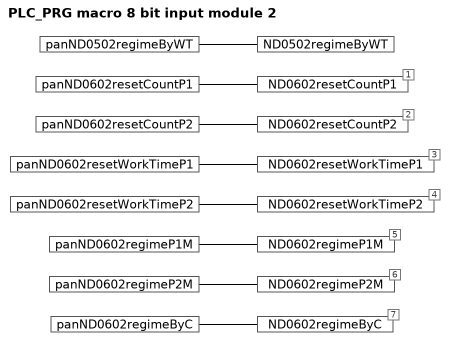
[picture p72: PLC_PRG macro 8 bit input module 2 (CFC)]
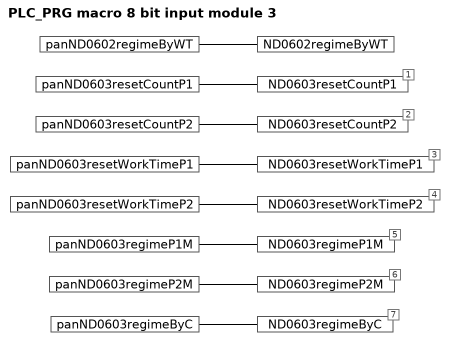
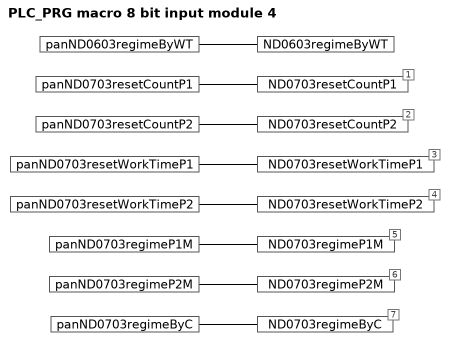
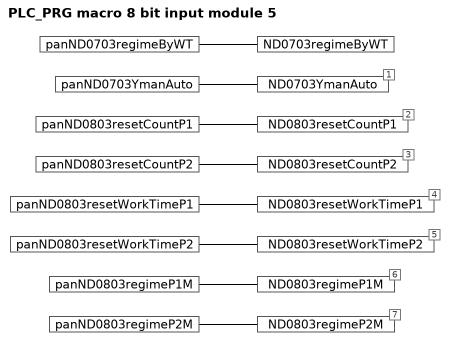
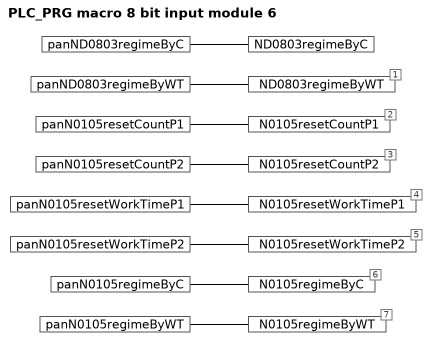
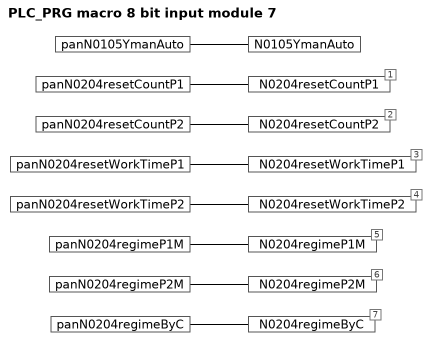
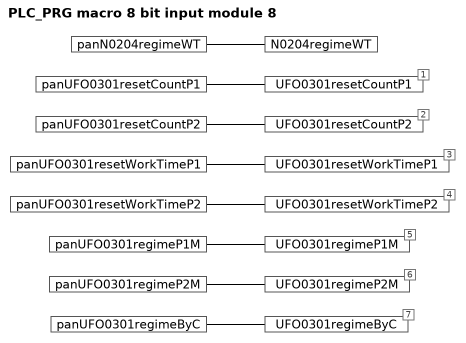
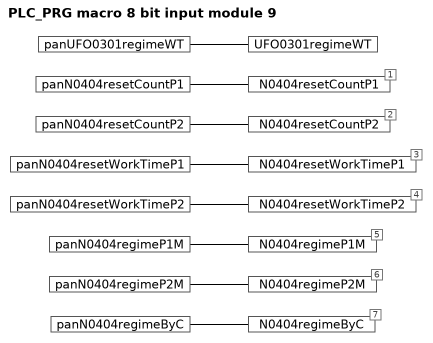
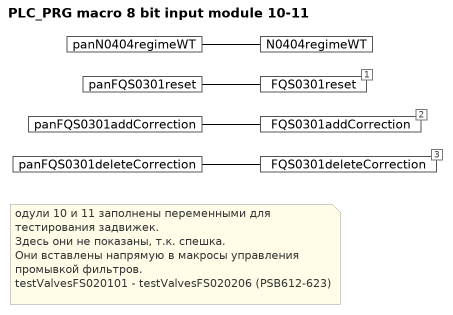
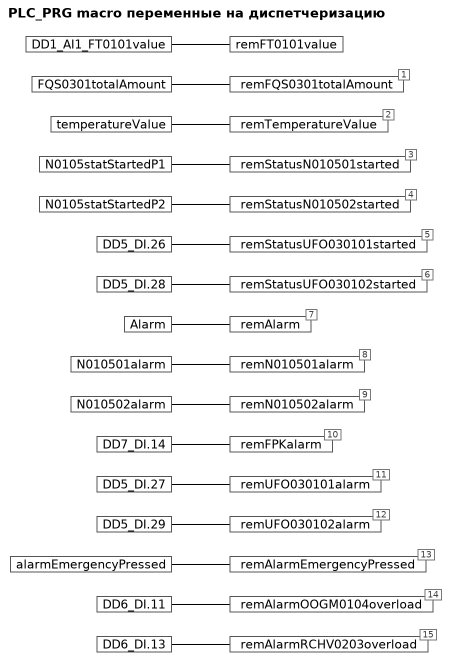
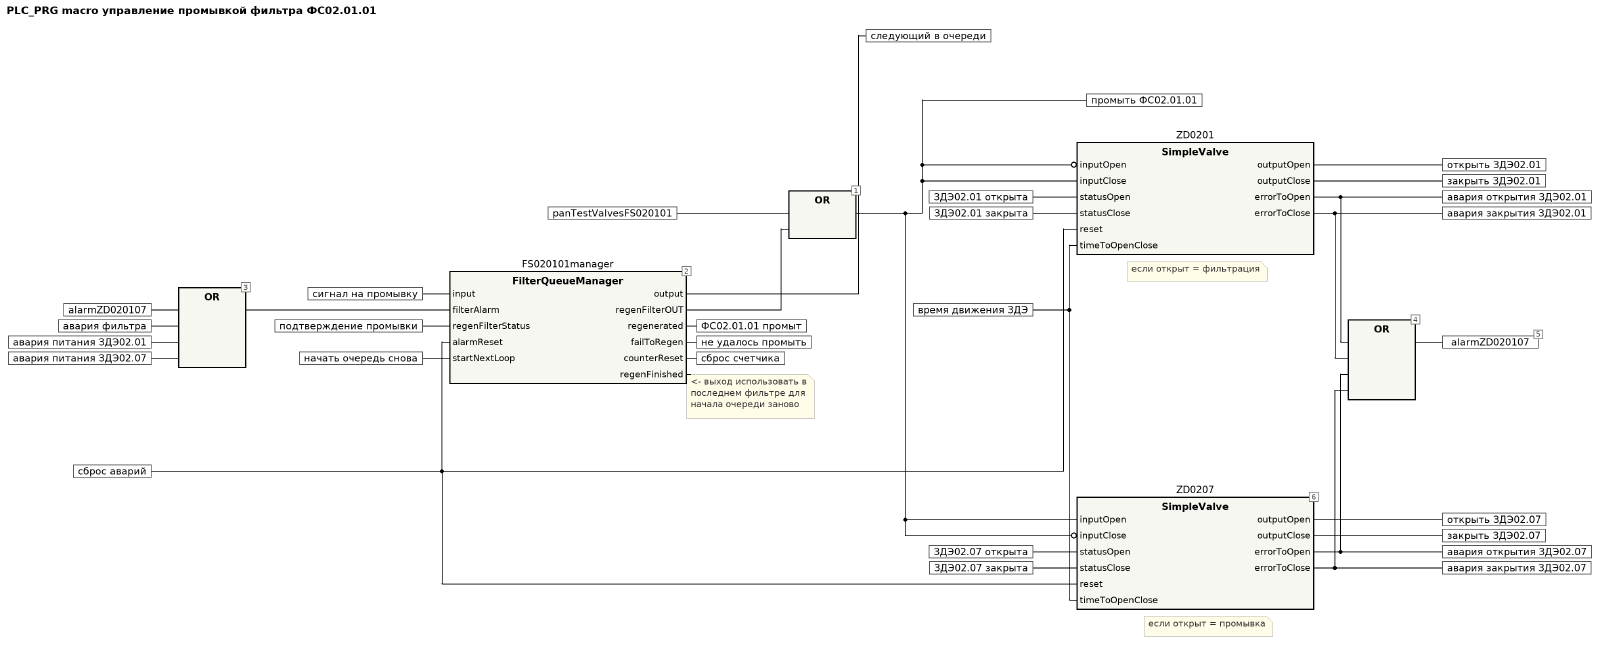
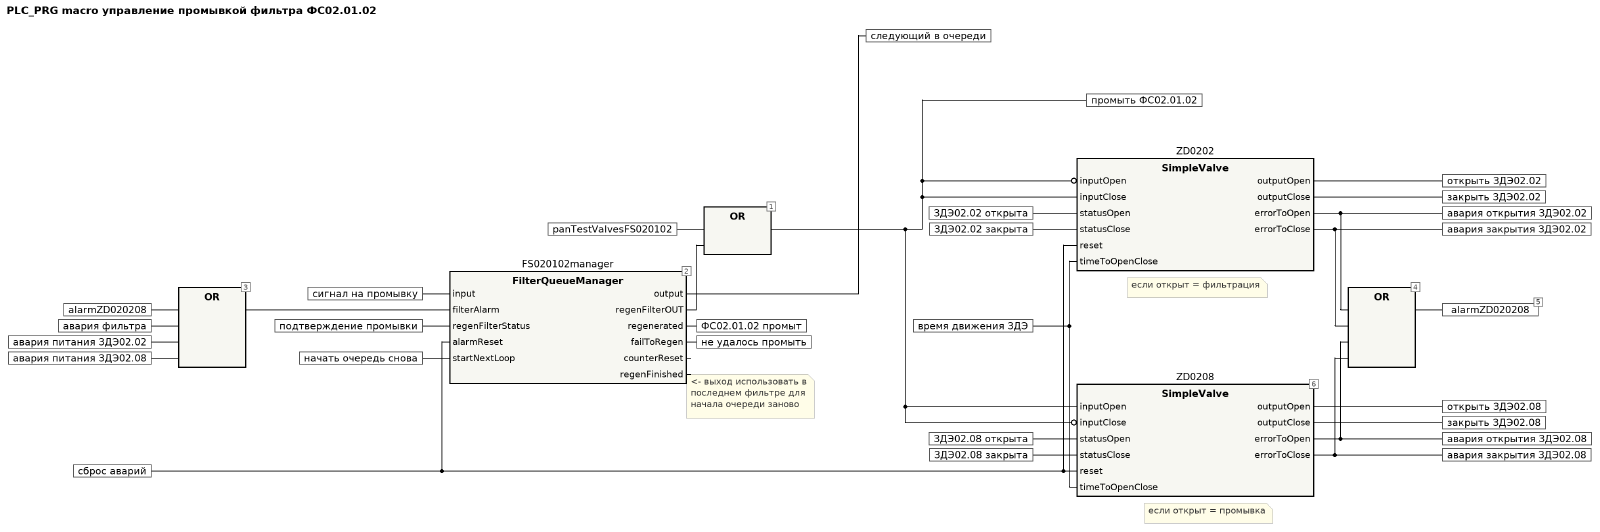
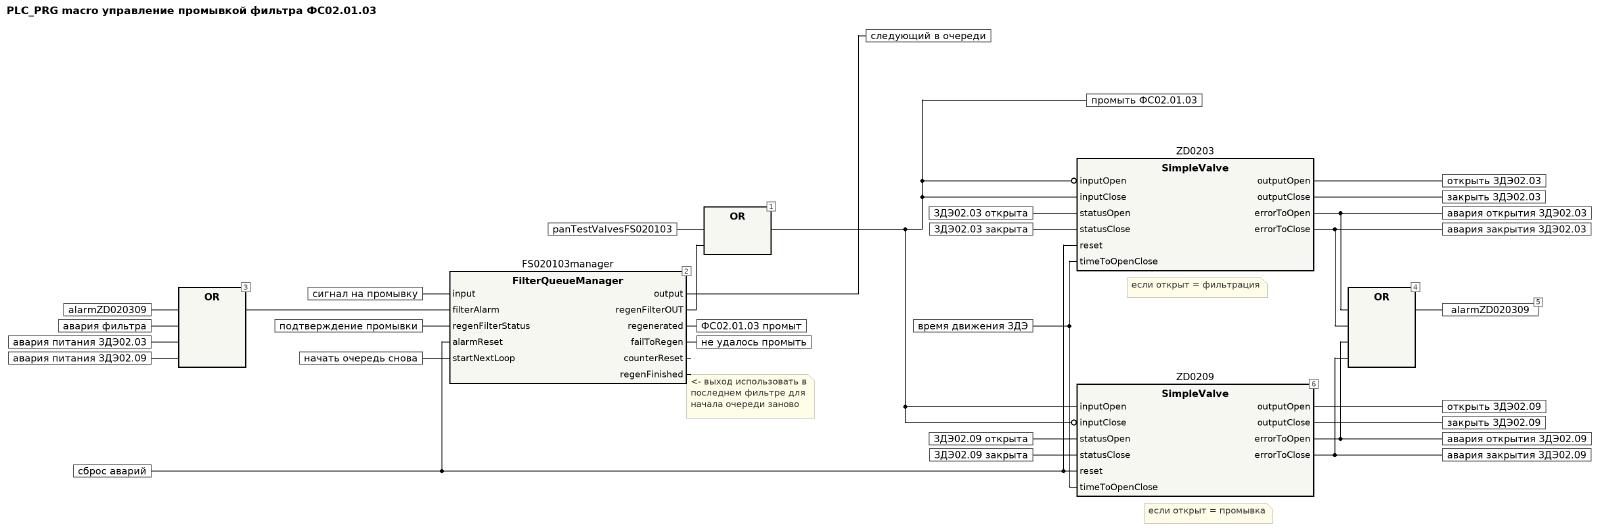
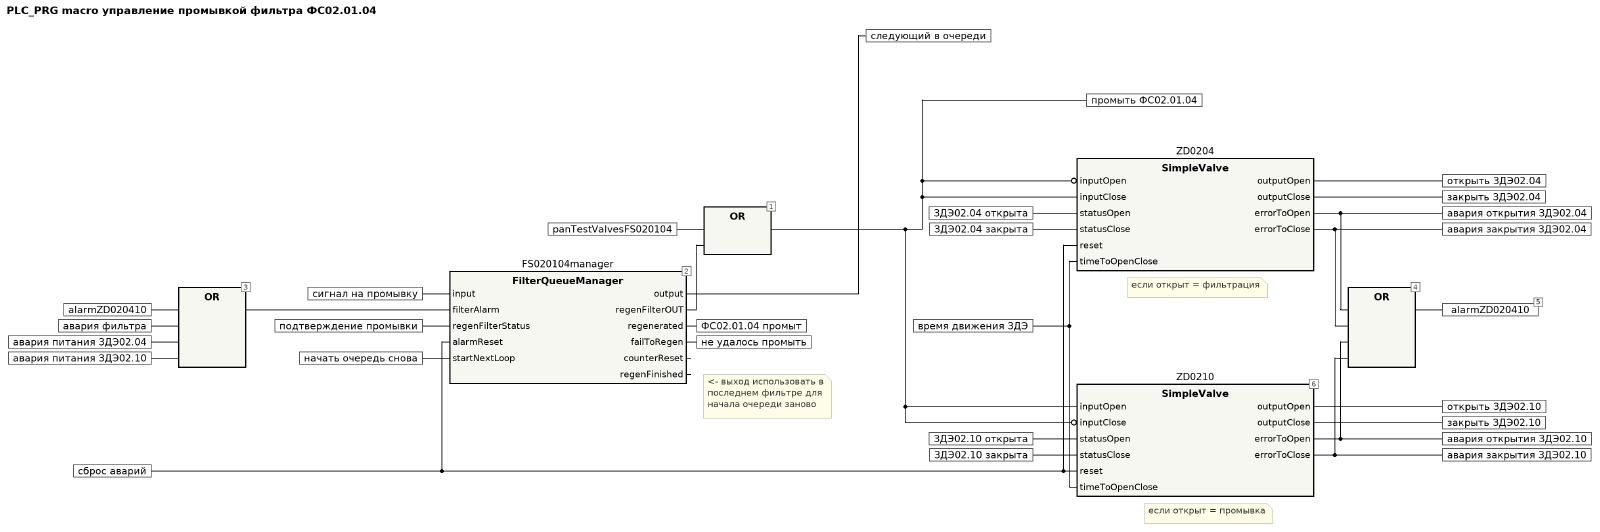
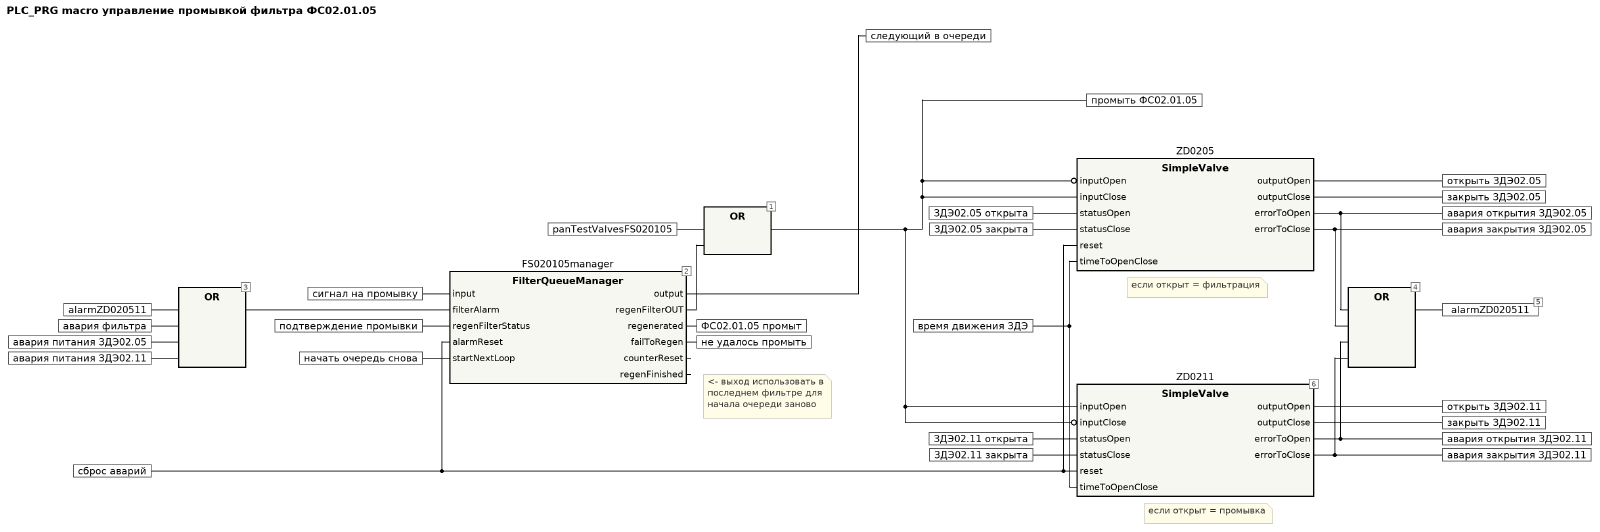
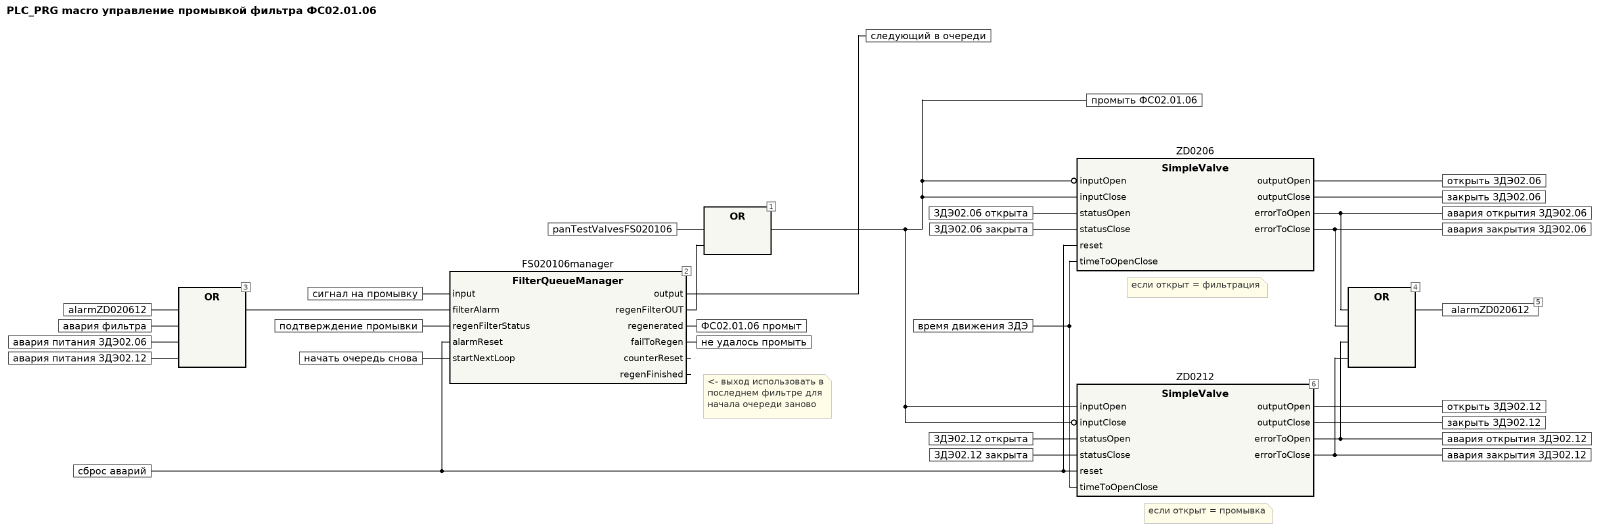
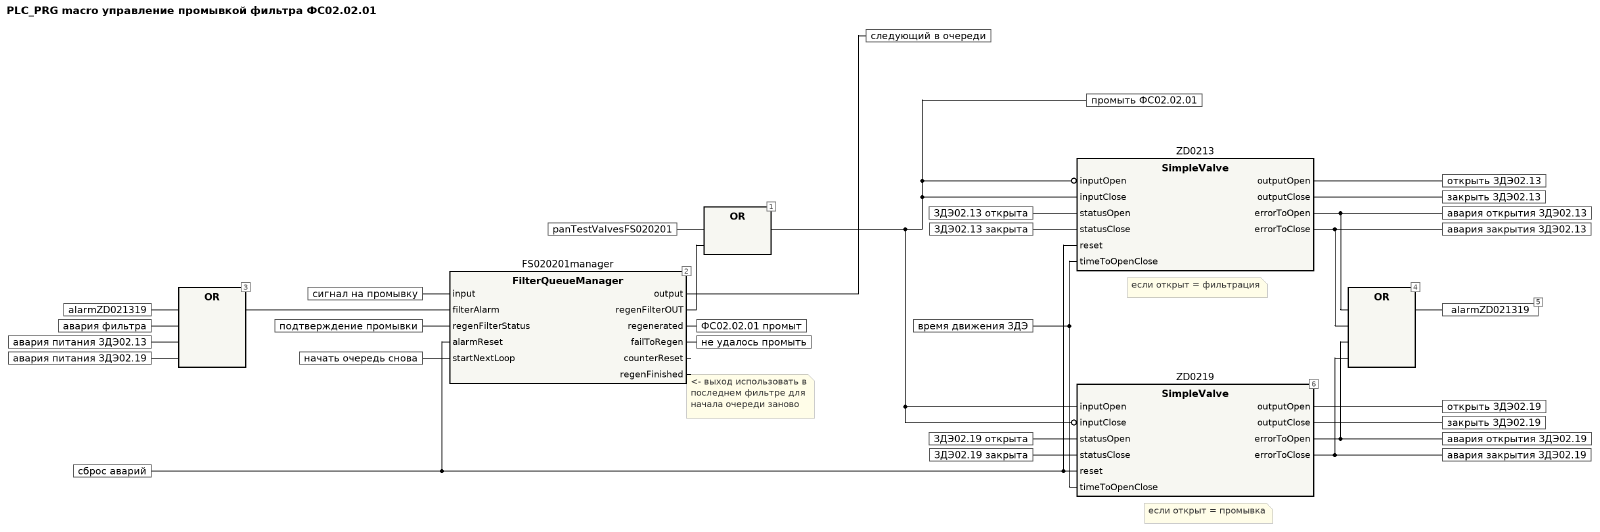
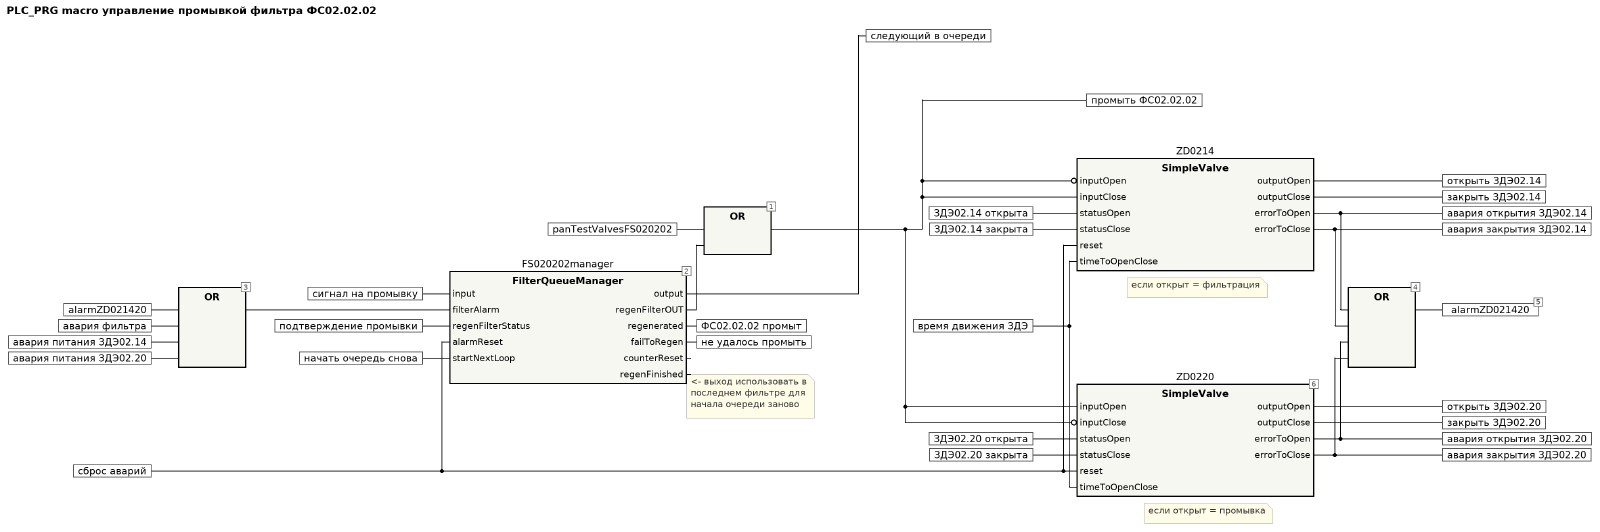
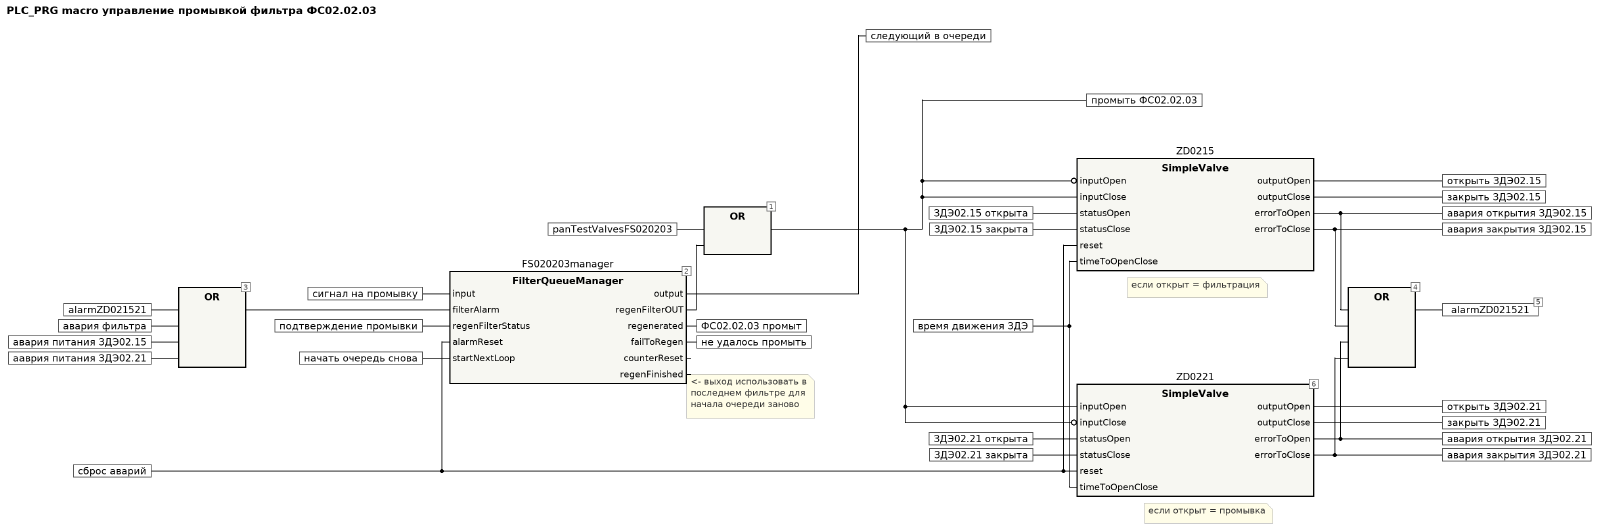
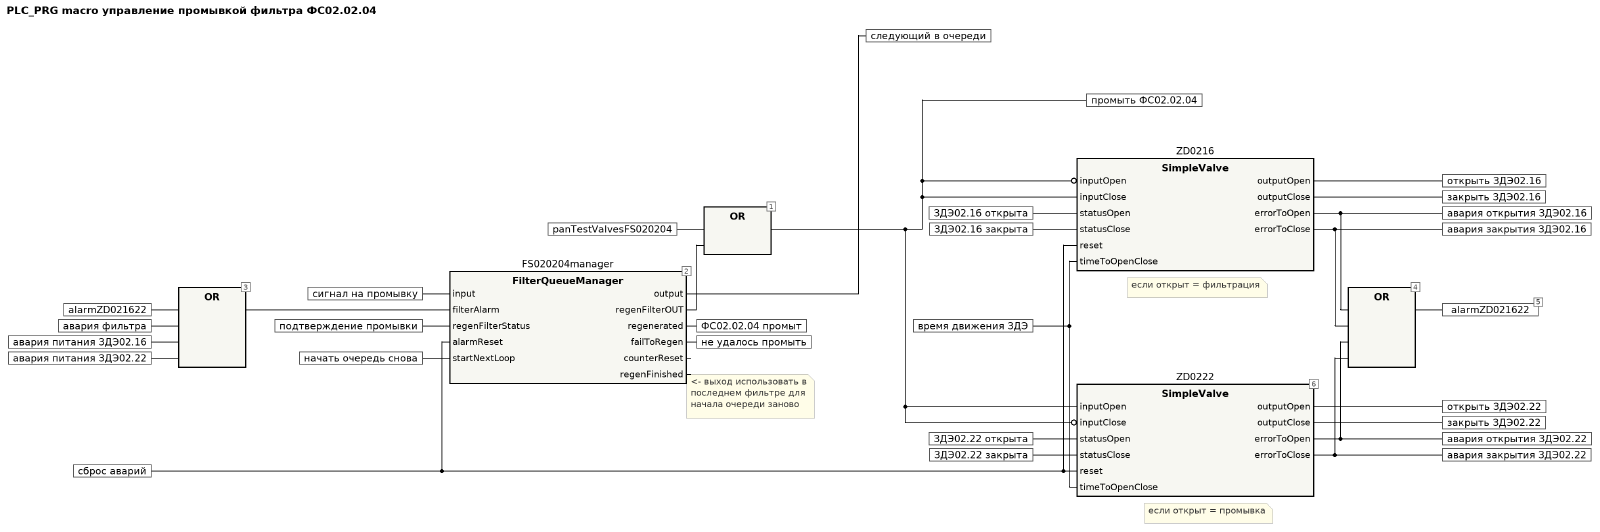
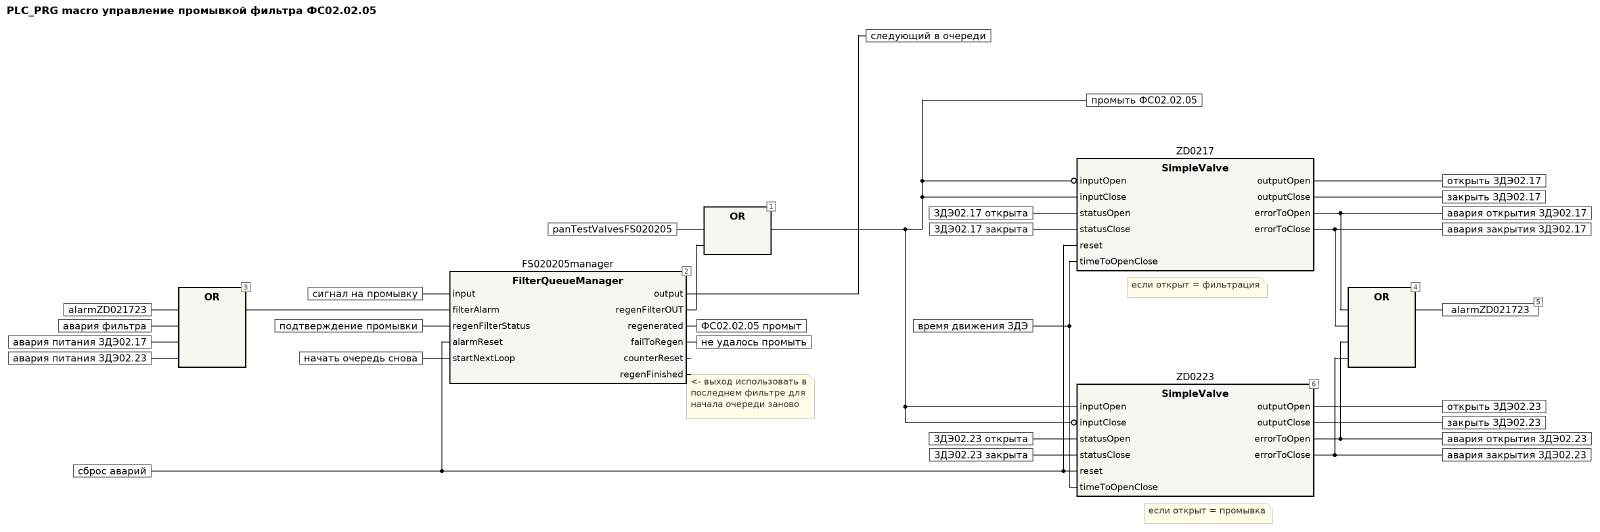
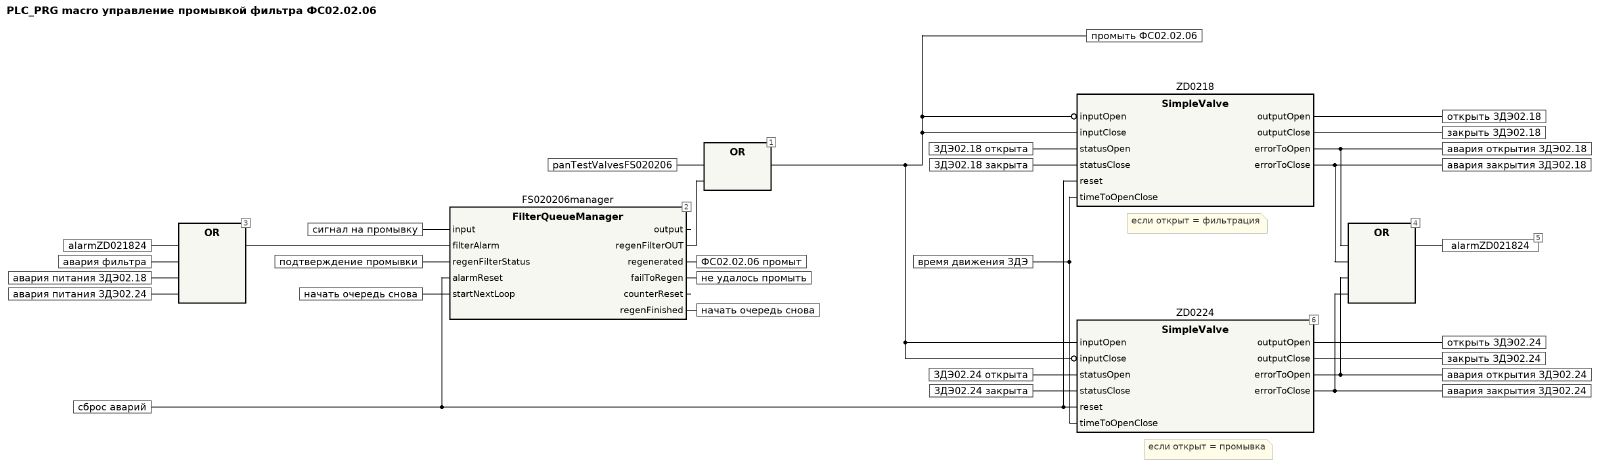
_CFC_ (* Continuous Function Chart, elements in execution order *)
(* в этом макросе лежит управление режимом тестирования задвижек ЗДЭ03 / Тестирование запрещает автоматический запуск УФО от ПЛК *)
(* 1=открыть; 0 = закрыть *)
(* авария питания КШЭ04.01 *)
(* авария НД05.02/02 *)
(* авария НД05.02/01 *)
(* инвертирование сигнала, чтобы все аварии / обозначались как 1 (TRUE) *)
(* авария питания ЗДЭ02.24 *)
(* авария питания ЗДЭ02.23 *)
(* авария питания ЗДЭ02.22 *)
(* авария питания ЗДЭ02.21 *)
(* авария питания ЗДЭ02.20 *)
(* авария питания ЗДЭ02.19 *)
(* авария питания ЗДЭ02.18 *)
(* авария питания ЗДЭ02.17 *)
(* авария питания ЗДЭ02.16 *)
(* авария питания ЗДЭ02.15 *)
(* авария питания ЗДЭ02.14 *)
(* авария питания ЗДЭ02.13 *)
(* авария питания ЗДЭ02.12 *)
(* авария питания ЗДЭ02.11 *)
(* авария питания ЗДЭ02.10 *)
(* авария питания ЗДЭ02.09 *)
(* авария питания ЗДЭ02.08 *)
(* авария питания ЗДЭ02.07 *)
(* авария питания ЗДЭ02.06 *)
(* авария питания ЗДЭ02.05 *)
(* авария питания ЗДЭ02.04 *)
(* авария питания ЗДЭ02.03 *)
(* авария питания ЗДЭ02.02 *)
(* авария питания ЗДЭ02.01 *)
(* очередь передается на 2 ступень *)
(* подсчет общего объема стоков, прошедшего через расходомер FT01.02 *)
(* сброс счетчика стоков до следующей промывки *)
(* авария (при 0) ФС02.02/01 *)
(* авария (при 0) ФС02.02/02 *)
(* авария (при 0) ФС02.02/03 *)
(* авария (при 0) ФС02.02/04 *)
(* авария (при 0) ФС02.02/05 *)
(* авария (при 0) ФС02.02/06 *)
(* авария (при 0) ФС02.01/01 *)
(* авария (при 0) ФС02.01/02 *)
(* авария (при 0) ФС02.01/03 *)
(* авария (при 0) ФС02.01/04 *)
(* авария (при 0) ФС02.01/05 *)
(* авария (при 0) ФС02.01/06 *)
(* 0=авария *)
(* заданный до промывки объем *)
(* текущий объем *)
(* Пуск Н02.04/02 *)
(* Пуск Н02.04/01 *)
(* Стоп Н02.04 *)
(* Сухой ход Н02.04 (LS02.03) 0=сух.ход *)
(* Клапан КЭМ08.01 открыт. *)
(* Клапан КЭМ07.01 открыт. *)
(* Клапан КЭМ06.01 открыт. *)
(* Клапан КЭМ05.01 открыт. *)
(* промывка ФС02.02/01 *)
(* промывка ФС02.02/02 *)
(* промывка ФС02.02/03 *)
(* промывка ФС02.02/04 *)
(* промывка ФС02.02/05 *)
(* промывка ФС02.02/06 *)
(* Авария Н02.04/02 (0=авария) *)
(* Авария Н02.04/01 (0=авария) *)
(* импульсный расходомер *)
(* авария Н04.04/02, 0=авария *)
(* авария Н04.04/01, 0=авария *)
(* сухой ход Н04.04, 0=защита *)
(* авт.пуск Н04.04 *)
(* пуск Н04.04/01 *)
(* пуск Н04.04/02 *)
(* стоп Н04.04 *)
(* подающий насос ФПК работает *)
(* статус КШЭ04.01 закрыт *)
(* Закрыть КШЭ04.01 *)
(* статус КШЭ04.01 открыт *)
(* Открыть КШЭ04.01 *)
(* авария ФПК *)
(* Авария входа AI6 ПЛК, давл.ФПК *)
(* Давление на входе ФПК / 0...16 бар (мах допуст.10) *)
(* LSА02.01 Перелив РЧВ02.03 *)
(* авария питания ЗДЭ02.25 *)
(* термоконтакт Н01.05/02 *)
(* термоконтакт Н01.05/01 *)
(* Авария ЧРП Н01.05 *)
(* КМ3 питание насоса 2 *)
(* КМ2 питание насоса 1 *)
(* КМ1 питание ЧРП *)
(* Пуск  Н01.05 *)
(* время на создание потока *)
(* Стоп  Н01.05 (сброс самоподхвата реле) *)
(* SA1 Ручной выбор Н01.05/02 = главный *)
(* SA1 Ручной выбор Н01.05/01 = главный *)
(* LS01.04 - нижний уровень ОГМ01.04, сухой ход Н01.05 *)
(* LS01.03 - рабочий верхний уровень ОГМ01.04 автоматический пуск 01.05 *)
(* Статус ПУСК ЧРП Н01.05 *)
(* Инициализирует требуемые булевые переменные / в момент старта выполнения программы. *)
(* LSA01.02 перелив ОГМ01.04 *)
(* сухой ход НД08.03/02 *)
(* сухой ход НД08.03/01 *)
(* сухой ход НД08.03/02 *)
(* сухой ход НД08.03/01 *)
(* авария входа рН-метра QE01.02 *)
(* рН-метр QE01.01 на входе, / диапазон 0...14 *)
(* расходомер FT01.02 на входе, / диапазон 0...600куб/час *)
(* авария входа расходомера FT01.01 *)
(* управление 4...20мА НД08.04 *)
(* пуск/стоп НД08.04 *)
(* насос Н04.01 работает *)
(* авария НД08.04 *)
(* авария привода НД08.03/02 *)
(* авария привода НД08.03/01 *)
(* АВАРИИ *)
(* управление 4...20мА НД05.02/02 *)
(* пуск/стоп НД05.02/02 *)
(* авария НД05.02/02 *)
(* авария НД05.02/01 *)
(* пуск/стоп НД05.02/01 *)
(* управление 4...20мА НД05.02/01 *)
(* датчик температуры в помещении / (метран) диапазон: 0...+100С *)
(* лампа АВАРИЯ *)
(* авария входа датчика температуры *)
(* ошибка блока дозирования НД05.02 *)
(* авария НД06.02/02 *)
(* авария НД06.02/01 *)
(* управление 4...20мА НД06.02/02 *)
(* пуск/стоп НД06.02/02 *)
(* пуск/стоп НД06.02/01 *)
(* управление 4...20мА НД06.02/01 *)
(* авария НД06.03/02 *)
(* авария НД06.03/01 *)
(* управление 4...20мА НД06.03/02 *)
(* пуск/стоп НД06.03/02 *)
(* пуск/стоп НД06.03/01 *)
(* управление 4...20мА НД06.03/01 *)
(* авария НД06.02/02 *)
(* авария НД06.02/01 *)
(* авария НД06.03/02 *)
(* авария НД06.03/01 *)
(* авария НД07.03/02 *)
(* авария НД07.03/01 *)
(* пуск/стоп НД07.03/02 *)
(* пуск/стоп НД07.03/01 *)
(* управление 4...20мА НД07.03/02 *)
(* управление 4...20мА НД07.03/01 *)
(* авария НД07.03/02 *)
(* авария НД07.03/01 *)
(* авария привода НД08.03/02 *)
(* авария привода НД08.03/01 *)
(* управление 4...20мА НД08.03/02 *)
(* пуск/стоп НД08.03/02 *)
(* пуск/стоп НД08.03/01 *)
(* управление 4...20мА НД08.03/01 *)
(* авария НД08.04 *)
(* расходомер FT01.01 на входе, / диапазон 0...600куб/час *)
(* авария входа расходомера FT01.02 *)
(* авария входа рН-метра QE01.01 *)
(* рН-метр QE01.02 на входе, / диапазон 0...14 *)
(* ФПК не запустился *)
(* ФПК готов к приему *)
(* подающий насос ФПК работает *)
(* авария ФПК *)
(* Давление на входе ФПК (0...16 бар) *)
(* датчик уровня осадка *)
(* Защита от сухого хода насоса ФПК *)
(* запуск фильтрации *)
(* время работы ФПК после спада сигнала датч.осадка *)
(* время контроля старта ФПК (по умолч.=3мин) *)
(* авария Н04.04/02 *)
(* авария Н04.04/01 *)
(* авария УФО03.01/01 *)
(* авария УФО03.01/02 *)
(* работа УФО03.01/01 *)
(* Для подачи предостережения на пульте / оператора (при необходимости), а также / сигнализации лампой АВАРИЯ. *)
(* авария УФО03.01/01 *)
(* работа УФО03.01/02 *)
(* авария УФО03.01/02 *)
(* Контроль, если УФО включили вручную, / а потока при этом нет. *)
(* работа М06.04 (УПК) *)
(* работа М07.02 (УПЩ) *)
(* работа М08.02 (УПФ) *)
(* авария М06.04 (УПК) *)
(* авария М07.02 (УПЩ) *)
(* авария М08.02 (УПФ) *)
(* пуск/стоп НД07.03/02 *)
(* пуск/стоп НД07.03/01 *)
(* пуск/стоп НД08.04 *)
(* пуск/стоп НД06.02/02 *)
(* пуск/стоп НД06.02/01 *)
(* пуск/стоп НД06.03/02 *)
(* пуск/стоп НД06.03/01 *)
(* пуск/стоп НД08.03/02 *)
(* пуск/стоп НД08.03/01 *)
(* промывка ФС02.01/01 *)
(* промывка ФС02.01/02 *)
(* промывка ФС02.01/03 *)
(* промывка ФС02.01/04 *)
(* промывка ФС02.01/05 *)
(* промывка ФС02.01/06 *)
(* Авария Н02.04/02 (0=авария) *)
(* Авария Н02.04/01 (0=авария) *)
(* здесь мгновенный расход / в кубометрах в час (FT01.02) *)
(* выдает импульс / каждую секунду *)
(* если есть расход / (больше нуля) *)
(* преобразуем расход из / кубометров в час в / кубометры в секунду *)
(* суммируем каждую секунду значение / мгновенного расхода в кубометрах в секунду *)
(* блок подачи сигнала на промывку *)
(* авария КНС *)
(* Авария питания розеток / управл.клапанов фильтров. *)
(* Авария питания клапанов КЭМ. *)
(* авария сети (РКФ) *)
(* Блок управления разрешением работы КНС *)
(* Нажат аварийный стоп. *)
(* разрешение работы КНС / 1 = разрешено *)
(* авария сети (РКФ) *)
(* Нажат аварийный стоп. *)
(* LSA01.02 перелив ОГМ01.04 *)
(* контроль обрыва или ошибок модулей в сети ПЛК *)
(* вкл КМ2 *)
(* статус-пуск Н01.05/01 *)
(* Статус ПУСК / ЧРП Н01.05 *)
(* вкл КМ3 *)
(* статус-пуск Н01.05/02 *)
(* авария питания ЗДЭ03.01 *)
(* авария питания ЗДЭ03.02 *)
(* авария обоих УФО, если проблемы / открытия/закрытия на одной из задвижек *)
(* 0 = перелив *)
#0 rTrigStartInitializer:R_TRIG(CLK: TRUE)
#1 startInitializer <= #0.Q
#2 MACRO контроль температуры в помещении(pin 1 "вход датчика температуры": DD1_AI0, pin 2 "минимально допустимая температура в помещении": maxTemperature, pin 3 "максимально допустимая температура в помещении": minTemperature)
	(* не смотрим конкретный тип ошибки / (работает не точно, обрыв определяет как слишком маленькое значение) / если не равно 0 - значит на входе ошибка *)
	(* задаем границы допустимой температуры в помещении / проверяем что измеренное значение в заданном диапазоне *)
	#3 DD1_AI0_temperature:DECODE_FLOAT(VALUE: pin 1, DEF_VALUE: -)
	#4 NE(#3._ERR, 0)
	out 2 "авария датчика температуры" <= #4
	out 1 "температура в помещении" <= #3.OUT_VALUE
	#5 REAL_TO_INT(#3.OUT_VALUE)
	#6 temperatureLimits:LIMITALARM(IN: #5, HIGH: pin 3, LOW: pin 2)
	out 3 "температура выше заданного диапазона" <= #6.O
	out 4 "температура ниже заданного диапазона" <= #6.U
	#7 temperatureLimits:LIMITALARM(IN: -, HIGH: -, LOW: -)
END_MACRO
#8 temperatureValue <= #2.out 1
#9 DD1_AI0_error <= #2.out 2
#10 alarmHighTemperature <= #2.out 3
#11 alarmLowTemperature <= #2.out 4
#12 OR(testKSHE0401, DD7_DI.13)
#13 MACRO клапан шаровый перед ФПК (КШЭ04.01)(pin 1 "сигнал "подающий насос ФПК" работает": #12, pin 2 "статус КШЭ04.01 открыт": DD9_DI.2, pin 3 "статус КШЭ04.01 закрыт": DD9_DI.3, pin 4 "сброс аварий": alarmReset, pin 5 "время на открытие/закрытие": timeToOpenCloseValve)
	#14 FPKkshe0401DelayToOpen:TON(IN: #16.outputOpen, PT: T#1s)
	out 1 "выход на открытие КШЭ04.01" <= #14.Q
	#15 FPKkshe0401DelayToClose:TON(IN: #16.outputClose, PT: T#1s)
	out 2 "выход на закрытие КШЭ04.01" <= #15.Q
	#16 FPKkshe0401:SimpleValve(inputOpen: pin 1, inputClose: #17, statusOpen: pin 2, statusClose: pin 3, reset: pin 4, timeToOpenClose: pin 5)
	#17 NOT(pin 1)
	out 3 "авария на открытие КШЭ04.01" <= #16.errorToOpen
	out 4 "авария на закрытие КШЭ04.01" <= #16.errorToClose
END_MACRO
#18 DD4_DO.2 <= #13.out 1
#19 DD4_DO.3 <= #13.out 2
#20 FPKkshe0401errorToOpen <= #13.out 3
#21 FPKkshe0401errorToClose <= #13.out 4
#22 OR(DD1_AI0_error, DD1_AI1_error, DD1_AI2_error, DD1_AI3_error, DD1_AI4_error, alarmHighTemperature, alarmLowTemperature, ND0502dosingError, ND0602dosingError, ND0603dosingError, ND0803dosingError, ND0804dosingError, DD1_DI6, DD1_DI7, N010501alarm, N010502alarm, ZDE0225errorToOpen, ZDE0225errorToClose, DD7_DI.14, FPKnotStarted, DD1_AI5_error, FPKkshe0401errorToOpen, FPKkshe0401errorToClose, DD5_DI.27, DD5_DI.29, filterFailToRegen020101, errorToOpenZD0201, errorToCloseZD0201, errorToOpenZD0207, errorToCloseZD0207, filterFailToRegen020102, errorToOpenZD0202, errorToCloseZD0202, errorToOpenZD0208, errorToCloseZD0208, filterFailToRegen020103, errorToOpenZD0203, errorToCloseZD0203, errorToOpenZD0209, errorToCloseZD0209, filterFailToRegen020104, errorToOpenZD0204, errorToCloseZD0204, errorToOpenZD0210, errorToCloseZD0210, filterFailToRegen020105, errorToOpenZD0205, errorToCloseZD0205, errorToOpenZD0211, errorToCloseZD0211, filterFailToRegen020106, errorToOpenZD0206, errorToCloseZD0206, errorToOpenZD0212, errorToCloseZD0212, filterFailToRegen020201, errorToOpenZD0213, errorToCloseZD0213, errorToOpenZD0219, errorToCloseZD0219, filterFailToRegen020202, errorToOpenZD0214, errorToCloseZD0214, errorToOpenZD0220, errorToCloseZD0220, filterFailToRegen020203, errorToOpenZD0215, errorToCloseZD0215, errorToOpenZD0221, errorToCloseZD0221, filterFailToRegen020204, errorToOpenZD0216, errorToCloseZD0216, errorToOpenZD0222, errorToCloseZD0222, filterFailToRegen020205, errorToOpenZD0217, errorToCloseZD0217, errorToOpenZD0223, errorToCloseZD0223, filterFailToRegen020206, errorToOpenZD0218, errorToCloseZD0218, errorToOpenZD0224, errorToCloseZD0224, alarmPLKnetwork, alarmND050201, alarmND050202, alarmND060201, alarmND060202, alarmND060301, alarmND060302, alarmND070301, alarmND070302, alarmND080301, alarmND080302, alarmND0804, alarmOGM0104overload, alarmRCHV0203overload, alarmN040402, alarmN040401, alarmM0604, alarmM0702, alarmM0802, alarmN020401, alarmN020402, alarmFS020101, alarmFS020102, alarmFS020103, alarmFS020104, alarmFS020105, alarmFS020106, alarmFS020201, alarmFS020202, alarmFS020203, alarmFS020204, alarmFS020205, alarmFS020206, alarmZDE0201power, alarmZDE0202power, alarmZDE0203power, alarmZDE0204power, alarmZDE0205power, alarmZDE0206power, alarmZDE0207power, alarmZDE0208power, alarmZDE0209power, alarmZDE0210power, alarmZDE0211power, alarmZDE0212power, alarmZDE0213power, alarmZDE0214power, alarmZDE0215power, alarmZDE0216power, alarmZDE0217power, alarmZDE0218power, alarmZDE0219power, alarmZDE0220power, alarmZDE0221power, alarmZDE0222power, alarmZDE0223power, alarmZDE0224power, alarmZDE0225power, alarmKSHE0401power, alarmKNS, alarmPowerSocketFS, alarmKEMvalvesPower, alarmEmergencyPressed, alarmRKF, errorToOpenZDE0301, errorToCloseZDE0301, errorToOpenZDE0302, errorToCloseZDE0302, alarmZDE0301power, alarmZDE0302power)
#23 DD1_DO11 <= #22
#24 alarm <= #22
#25 MACRO контроль аналогового входа DD1_AI1(pin 1 "вход": DD1_AI1)
	(* Не смотрим конкретную ошибку, / определяем,что вход неисправен без расшифровки. *)
	#26 DD1_AI1_FT0101:DECODE_FLOAT(VALUE: pin 1, DEF_VALUE: -)
	#27 NE(#26._ERR, 0)
	out 2 "авария" <= #27
	out 1 "выход" <= #26.OUT_VALUE
END_MACRO
#28 DD1_AI1_FT0101value <= #25.out 1
#29 DD1_AI1_error <= #25.out 2
#30 MACRO контроль аналогового входа DD1_AI2(pin 1 "вход": DD1_AI2)
	(* Не смотрим конкретную ошибку, / определяем,что вход неисправен без расшифровки. *)
	#31 DD1_AI2_FT0102:DECODE_FLOAT(VALUE: pin 1, DEF_VALUE: -)
	#32 NE(#31._ERR, 0)
	out 2 "авария" <= #32
	out 1 "выход" <= #31.OUT_VALUE
END_MACRO
#33 DD1_AI2_FT0102value <= #30.out 1
#34 DD1_AI2_error <= #30.out 2
#35 MACRO управление Н01.05 (поддержание заданного расхода по FT01.02)(pin 1 "статус ПУСК ЧРП (реле)": DD5_DI.4, pin 2 "LS01.03 раб.уров.": DD6_DI.12, pin 3 "LS01.04 ниж.уров.(сух.ход)": DD5_DI.0, pin 4 "SA1ручной выб.Н01.05/01-главный": DD5_DI.5, pin 5 "SA1ручной выб.Н01.05/02-главный": DD5_DI.6, pin 6 "включить режим "по кол.вкл."": N0105regimeByC, pin 7 "включить режим "по наработке"": N0105regimeByWT, pin 8 "значение расхода от FT01.02": DD1_AI2_FT0102value, pin 9 "уставка расхода": N0105flowSetValue, pin 10 "время на создание потока": N0105minFlowTime, pin 11 "Р-коэфф.": N0105koeffP, pin 12 "I-коэфф": N0105koeffI, pin 13 "Д-коэфф": N0105koeffD, pin 14 "управление ЧРП в ручн.реж.(4...20мА)": N0105YoutManual, pin 15 "переключатель управление ЧРП РУЧН/АВТ": N0105YmanAuto, pin 16 "мин.допустимый расход": N0105minFlow, pin 17 "термоконтакт Н01.05/01": DD5_DI.2, pin 18 "термоконтакт Н01.05/02": DD5_DI.3, pin 19 "авария ЧРП Н01.05": DD5_DI.1, pin 20 "сброс аварии": alarmReset, pin 21 "сброс кол-ва вкл.Н01.05/01": N0105resetCountP1, pin 22 "сброс кол-ва вкл.Н01.05/02": N0105resetCountP2, pin 23 "сброс наработки Н01.05/01": N0105resetWorkTimeP1, pin 24 "сброс наработки Н01.05/02": N0105resetWorkTimeP2)
	(* Если насос создает давление меньше / указанного, то авария. *)
	(* если на входе true / то нижнее значение, / иначе то, что посередине *)
	(* по умолчанию при старте программы *)
	(* управление Н01.05 - поддержание / заданного расхода по FT01.02 *)
	(* режимы по количеству включений,  или по наработке / активны если оба входа SA1 не активны *)
	(* Пуск  Н01.05 *)
	(* время на создание потока *)
	#36 OR(pin 2, #37.Q)
	#37 N0105startTrig:R_TRIG(CLK: pin 1)
	#38 N0105stopTrig:F_TRIG(CLK: pin 1)
	#39 N0105startTrigg:RS(SET: #36, RESET1: #41)
	#40 N0105regime:choosePumpRegime(start: #39.Q1, pump1Main: pin 4, pump2Main: pin 5, byCounter: #45, byWorkTime: #54)
	out 2 "статус режим "Н01.05/01 - главный"" <= #40.pump1MainActive
	out 3 "статус режим "Н01.05/02 - главный"" <= #40.pump2MainActive
	out 4 "статус режим "по кол-ву вкл."" <= #40.byCounterActive
	#41 OR(#38.Q, #42)
	out 5 "статус режим "по наработке"." <= #40.byWorkTimeActive
	#42 NOT(pin 3)
	#43 NOT(#39.Q1)
	out 1 "СТОП (сброс самоподхвата реле пуска ЧРП)." <= #43
	#44 AND(#53.pump1active, #63)
	out 15 "авария Н01.05/01" <= #47.Q1
	#45 AND(NOT pin 4, NOT pin 5, #51.Q1)
	#46 OR(#44, #52, NOT pin 17)
	#47 N010501alarmTrig:RS(SET: #46, RESET1: pin 20)
	#48 N010501alarm <= #47.Q1
	#49 OR(pin 6, startInitializer)
	#50 N0105regByCinit:R_TRIG(CLK: #49)
	#51 N0105regByCtrig:RS(SET: #50.Q, RESET1: #55.Q)
	#52 AND(#53.pump1active, NOT pin 19)
	#53 N0105twoPumpOneDriveManager:TwoPumpOneDriveManager(startStopPump1: #40.startPump1, startStopPump2: #40.startPump2, alarmPump1: N010501alarm, alarmPump2: N010502alarm, alarmReset: alarmReset, counterStart: #40.startByCounter, Pump1ResetCounter: pin 21, Pump2ResetCounter: pin 22, ValueToResetCounter: -, workTimeStart: #40.startByWorkTime, workTimePump1Reset: pin 23, workTimePump2Reset: pin 24, timeKM1off: -, timeKM23DelayON: -, timeKM23offDelay: -, timeReadyToStartDelay: -)
	out 6 "кол-во включений Н01.05/01" <= #53.counterPump1
	out 7 "кол-во включений Н01.05/02" <= #53.counterPump2
	out 8 "наработка Н01.05/01" <= #53.currentWorkTimePump1
	#54 AND(NOT pin 4, NOT pin 5, #56.Q1)
	out 9 "наработка Н01.05/02" <= #53.currentWorkTimePump2
	out 10 "КМ1-питание ЧРП" <= #53.DriveKM
	#55 N0105regWTinit:R_TRIG(CLK: pin 7)
	#56 N0105regWTtrig:RS(SET: #55.Q, RESET1: #50.Q)
	out 11 "КМ2-питание Н01.05/01" <= #53.pump1KM
	out 12 "КМ3-питание Н01.05/02" <= #53.pump2KM
	out 13 "пуск ЧРП (Н01.05)" <= #53.driveStart
	out 16 "авария Н01.05/02" <= #59.Q1
	#57 AND(NOT pin 19, #53.pump2active)
	#58 OR(#57, #61, NOT pin 18)
	#59 N010502alarmTrig:RS(SET: #58, RESET1: pin 20)
	#60 N010502alarm <= #59.Q1
	#61 AND(#53.pump2active, #63)
	#62 N0105timerminFlow:TON(IN: #53.driveStart, PT: pin 10)
	#63 AND(#62.Q, #64)
	#64 LE(pin 8, pin 16)
	#65 SEL(#53.driveStart, 0, #66.Y)
	out 14 "управление ЧРП (4...20мА)" <= #65
	#66 N0105pidReg:PID(ACTUAL: pin 8, SET_POINT: pin 9, KP: pin 11, TN: pin 12, TV: pin 13, Y_MANUAL: pin 14, Y_OFFSET: -, Y_MIN: 4, Y_MAX: 20, MANUAL: pin 15, RESET: #66.OVERFLOW)
END_MACRO
#67 DD4_DO.13 <= #35.out 1
#68 N0105statRegimeP1M <= #35.out 2
#69 N0105statRegimeP2M <= #35.out 3
#70 N0105statRegimeByC <= #35.out 4
#71 N0105statRegimeByWT <= #35.out 5
#72 N0105counterP1 <= #35.out 6
#73 N0105counterP2 <= #35.out 7
#74 N0105workTimeP1 <= #35.out 8
#75 N0105workTimeP2 <= #35.out 9
#76 DD2_DO.0 <= #35.out 10
#77 DD2_DO.1 <= #35.out 11
#78 DD2_DO.2 <= #35.out 12
#79 DD1_DO0 <= #35.out 13
#80 DD1_AO0 <= #35.out 14
#81 N010501alarm <= #35.out 15
#82 N010502alarm <= #35.out 16
#83 MACRO Сигналы работы с ФП04.02 (фильтр-пресс)(pin 1 "датчик уровня осадка": DD7_DI.15, pin 2 "время работы ФПК (после выкл.датч.осадка)": FPKtimeToWork, pin 3 "защита от сухого хода": DD6_DI.10, pin 4 "ошибка входа AI (обрыв)": DD1_AI5_error, pin 5 "авария ФПК": DD7_DI.14, pin 6 "фильтр-пресс готов к приему": DD7_DI.12, pin 7 "давление на входе в ФПК": DD1_AI5_FPKpressureValue, pin 8 "мах допустимое давление": FPKmaxPressureValue, pin 9 "подающий насос ФПК работает": DD7_DI.13, pin 10 "время контроля старта ФПК": FPKnotStartedTime, pin 11 "сброс аварий": alarmReset)
	(* Условие сброса сигнала о грязном фильтр-прессе: / 1. Пропал сигнал о готовности ФПК; / 2. Появился сигнал о готовности ФПК. / Это значит, что оператор раздвигал плиты, / чистил и снова сдвигал их. *)
	(* максимально допустимое давление / на входе ФПК *)
	(* Давление на входе ФПК / 0...16 бар (мах допуст.10) *)
	(* Время работы ФПК после / спада сигнала уровня осадка / по умолч.15мин. *)
	(* LES01.01-сигнал датчика уровня осадка ОГМ01.04 / запуск процесса фильтрации *)
	(* LS01.01-нижн.уровень на входе ОГМ01.04 / защита от сух. хода насоса ФПК *)
	(* ФПК готов к приему осадка *)
	#84 FPKneedToCleanResetFtrig:F_TRIG(CLK: FPKneedToCleanReset)
	#85 FPKstartTrig:RS(SET: pin 1, RESET1: #91)
	out 1 "запуск/старт ФПК" <= #85.Q1
	#86 FPKstopTimer:TOF(IN: pin 1, PT: pin 2)
	#87 FPKstopFtrig:F_TRIG(CLK: #86.Q)
	#88 AND(#85.Q1, #89)
	#89 NOT(pin 11)
	#90 AND(#85.Q1, #92.Q, #94)
	out 2 "ФПК не стартовал" <= #90
	#91 OR(#87.Q, pin 4, pin 5, #93, #95, #98.Q1)
	#92 FPKnotStartedTimer:TON(IN: #88, PT: pin 10)
	#93 NOT(pin 3)
	#94 NOT(pin 9)
	#95 NOT(pin 6)
	#96 AND(#85.Q1, #97)
	#97 GE(pin 7, pin 8)
	#98 FPKneedToCleanTrig:RS(SET: #96, RESET1: #84.Q)
	out 3 "ФПК нужно почистить!" <= #98.Q1
	#99 S FPKneedToCleanReset <= #98.Q1
	#100 FPKneedToCleanResetRtrig:R_TRIG(CLK: pin 6)
	#101 R FPKneedToCleanReset <= #100.Q
END_MACRO
#102 DD1_DO10 <= #83.out 1
#103 FPKnotStarted <= #83.out 2
#104 FPKneedToClean <= #83.out 3
#105 MACRO контроль аналогового входа DD1_AI3(pin 1 "вход": DD1_AI3)
	(* Не смотрим конкретную ошибку, / определяем,что вход неисправен без расшифровки. *)
	#106 DD1_AI3_QE0101:DECODE_FLOAT(VALUE: pin 1, DEF_VALUE: -)
	#107 NE(#106._ERR, 0)
	out 2 "авария" <= #107
	out 1 "выход" <= #106.OUT_VALUE
END_MACRO
#108 DD1_AI3_QE0101value <= #105.out 1
#109 DD1_AI3_error <= #105.out 2
#110 MACRO контроль аналогового входа DD1_AI4(pin 1 "вход": DD1_AI4)
	(* Не смотрим конкретную ошибку, / определяем,что вход неисправен без расшифровки. *)
	#111 DD1_AI4_QE0102:DECODE_FLOAT(VALUE: pin 1, DEF_VALUE: -)
	#112 NE(#111._ERR, 0)
	out 2 "авария" <= #112
	out 1 "выход" <= #111.OUT_VALUE
END_MACRO
#113 DD1_AI4_QE0102value <= #110.out 1
#114 DD1_AI4_error <= #110.out 2
#115 MACRO контроль аналогового входа DD1_AI5(pin 1 "вход": DD1_AI5)
	(* Не смотрим конкретную ошибку, / определяем,что вход неисправен без расшифровки. *)
	#116 DD1_AI5_FPK:DECODE_FLOAT(VALUE: pin 1, DEF_VALUE: -)
	#117 NE(#116._ERR, 0)
	out 2 "авария" <= #117
	out 1 "выход" <= #116.OUT_VALUE
END_MACRO
#118 DD1_AI5_FPKpressureValue <= #115.out 1
#119 DD1_AI5_error <= #115.out 2
#120 MACRO управление НД05.02 УПГ(pin 1 "вход расходомера в куб/час": DD1_AI1_FT0101value, pin 2 "max производительность НД в мл/мин": ND0502setMaxDosVal, pin 3 "задание дозирования в мл/куб": ND0502setKoefProp, pin 4 "режим:1 насос главный": ND0502regimeP1M, pin 5 "режим: 2 насос главный": ND0502regimeP2M, pin 6 "режим: по наработке": ND0502regimeByWT, pin 7 "режим: по кол-ву включений": ND0502regimeByC, pin 8 "авария 1 насоса": DD6_DI.0, pin 9 "авария 2 насоса": DD6_DI.1, pin 10 "сброс аварий": alarmReset, pin 11 "сброс счетчика включений 1 насоса": ND0502resetCountP1, pin 12 "сброс ссчетчика включений 2 насоса": ND0502resetCountP2, pin 13 "сброс наработки 1 насоса": ND0502resetWorkTimeP1, pin 14 "сброс наработки 2 насоса": ND0502resetWorkTimeP2)
	(* Если на входе SEL = TRUE, / то нижнее значение, / иначе - то,что посередине. *)
	(* сигнал 4...20мА на НД05.02/01 *)
	(* сигнал 4...20мА на НД05.02/02 *)
	#121 SEL(#128.pump1ON, 4, #122.outputValue)
	out 6 "выход 4...20мА насоса 1" <= #121
	#122 ND0502dosing:DosingPumpProportional(flowValue: pin 1, setMinPumpDosingValue: -, setMaxPumpDosingValue: pin 2, minOutputValue: -, maxOutputValue: -, setKoeffProportionality: pin 3, minFlowToStart: -)
	out 1 "ошибка блока дозирования" <= #122.dosingError
	#123 SEL(#128.pump2ON, 4, #122.outputValue)
	#124 linTrafo050202:LIN_TRAFO(IN: #123, IN_MIN: 4, IN_MAX: 20, OUT_MIN: 0, OUT_MAX: 1000)
	#125 REAL_TO_WORD(#124.OUT)
	out 7 "выход 4...20мА насоса 2" <= #125
	#126 ND0502regime:choosePumpRegime(start: #122.startDosingPump, pump1Main: pin 4, pump2Main: pin 5, byCounter: #127, byWorkTime: pin 6)
	out 2 "статус: 1 насос главный" <= #126.pump1MainActive
	out 3 "статус: 2 насос главный" <= #126.pump2MainActive
	out 4 "статус: по кол-ву включений" <= #126.byCounterActive
	#127 OR(pin 7, startInitializer)
	out 5 "статус: по наработке" <= #126.byWorkTimeActive
	#128 ND0502manager:TwoPumpManager(startStopPump1: #126.startPump1, startStopPump2: #126.startPump2, alarmPump1: #129, alarmPump2: #130, alarmReset: pin 10, counterStart: #126.startByCounter, Pump1ResetCounter: pin 11, Pump2ResetCounter: pin 12, ValueToResetCounter: -, workTimeStart: #126.startByWorkTime, workTimePump1Reset: pin 13, workTimePump2Reset: pin 14)
	out 12 "сигнал на включение насоса 1" <= #128.pump1ON
	#129 NOT(pin 8)
	out 13 "сигнал на включение насоса 2" <= #128.pump2ON
	out 8 "счетчик включений насоса 1" <= #128.counterPump1
	#130 NOT(pin 9)
	out 9 "счетчик включений насоса 2" <= #128.counterPump2
	out 10 "счетчик наработки насоса 1" <= #128.currentWorkTimePump1
	out 11 "счетчик наработки насоса 2" <= #128.currentWorkTimePump2
END_MACRO
#131 ND0502dosingError <= #120.out 1
#132 ND0502statRegimeP1M <= #120.out 2
#133 ND0502statRegimeP2M <= #120.out 3
#134 ND0502statRegimeByC <= #120.out 4
#135 ND0502statRegimeByWT <= #120.out 5
#136 DD1_AO3 <= #120.out 6
#137 DD10_AO0 <= #120.out 7
#138 ND0502counterP1 <= #120.out 8
#139 ND0502counterP2 <= #120.out 9
#140 ND0502workTimeP1 <= #120.out 10
#141 ND0502workTimeP2 <= #120.out 11
#142 DD4_DO.4 <= #120.out 12
#143 DD4_DO.5 <= #120.out 13
#144 AND(DD2_DO.1, DD5_DI.4)
#145 N0105statStartedP1 <= #144
#146 AND(DD5_DI.4, DD2_DO.2)
#147 N0105statStartedP2 <= #146
#148 MACRO Наполнение РЧВ02.03 (заслонка ЗДЭ02.25)(pin 1 "LS02.02раб.верх.уровень РЧВ": DD6_DI.14, pin 2 "LSA02.01 Перелив РЧВ": DD6_DI.13, pin 3 "статус ЗДЭ02.25 открыт": DD9_DI.0, pin 4 "статус ЗДЭ02.25 закрыт": DD9_DI.1, pin 5 "сброс аварий": alarmReset, pin 6 "время на открытие/закрытие": timeToOpenCloseValve)
	#149 OR(testZDE0225, pin 1)
	#150 NOT(pin 1)
	#151 ZDE0225:SimpleValve(inputOpen: #149, inputClose: #152, statusOpen: pin 3, statusClose: pin 4, reset: pin 5, timeToOpenClose: pin 6)
	out 1 "выход на открытие ЗДЭ02.25" <= #151.outputOpen
	#152 OR(#150, #153)
	out 2 "выход на закрытие ЗДЭ02.25" <= #151.outputClose
	out 3 "авария на открытие ЗДЭ02.25" <= #151.errorToOpen
	#153 NOT(pin 2)
	out 4 "авария на закрытие ЗДЭ02.25" <= #151.errorToClose
END_MACRO
#154 DD4_DO.0 <= #148.out 1
#155 DD4_DO.1 <= #148.out 2
#156 ZDE0225errorToOpen <= #148.out 3
#157 ZDE0225errorToClose <= #148.out 4
#158 MACRO управление Н02.04 (подача из РЧВ)(pin 1 "промывка ФС02.01/01": DD6_DI.20, pin 2 "промывка ФС02.01/02": DD6_DI.22, pin 3 "промывка ФС02.01/03": DD6_DI.24, pin 4 "промывка ФС02.01/04": DD6_DI.26, pin 5 "промывка ФС02.01/05": DD6_DI.28, pin 6 "промывка ФС02.01/06": DD6_DI.30, pin 7 "промывка ФС02.02/01": DD7_DI.0, pin 8 "промывка ФС02.02/02": DD7_DI.2, pin 9 "промывка ФС02.02/03": DD7_DI.4, pin 10 "промывка ФС02.02/04": DD7_DI.6, pin 11 "промывка ФС02.02/05": DD7_DI.8, pin 12 "промывка ФС02.02/06": DD7_DI.10, pin 13 "открыт КЭМ05.01": DD1_DI11, pin 14 "открыт КЭМ06.01": DD1_DI10, pin 15 "открыт КЭМ07.01": DD1_DI9, pin 16 "открыт КЭМ08.01": DD1_DI8, pin 17 "сухой ход Н02.04 (0=сух.ход)": DD5_DI.11, pin 18 "выбрать режим: Н02.04/01 - главный": N0204regimeP1M, pin 19 "выбрать режим: Н02.04/02 - главный": N0204regimeP2M, pin 20 "выбрать режим: по кол-ву включений": N0204regimeByC, pin 21 "выбрать режим: по наработке": N0204regimeWT, pin 22 "авария Н02.04/01 (0=авария)": DD5_DI.7, pin 23 "авария Н02.04/02 (0=авария)": DD5_DI.8, pin 24 "сброс аварий": alarmReset, pin 25 "сброс счетчика включений Н02.04/01": N0204resetCountP1, pin 26 "сброс счетчика включений Н02.04/02": N0204resetCountP2, pin 27 "сброс счетчика наработки Н02.04/01": N0204resetWorkTimeP1, pin 28 "сброс счетчика наработки Н02.04/02": N0204resetWorkTimeP2)
	(* Защита от сухого хода Н02.04 / (LS02.03) 0=сух.ход *)
	(* сброс самоподхвата реле *)
	(* Контроль открытия хотя бы одного из клапанов КЭМ *)
	(* Удержание сигнала на выключение насосов для / гарантированного сброса самоподхвата реле. *)
	(* Проверка, что фильтры 2 / ступени в регенерации (промывке) *)
	(* Проверка, что фильтры 1 / ступени в регенерации (промывке) *)
	#159 OR(pin 1, pin 2, pin 3, pin 4, pin 5, pin 6)
	#160 OR(#159, #161, #162)
	#161 OR(pin 7, pin 8, pin 9, pin 10, pin 11, pin 12)
	#162 OR(pin 13, pin 14, pin 15, pin 16)
	#163 N020401fTrigStop:F_TRIG(CLK: #170.pump1ON)
	#164 AND(#160, pin 17)
	#165 OR(#163.Q, #168.Q)
	#166 N0204stop:TOF(IN: #165, PT: T#1s)
	out 5 "стоп Н02.04" <= #166.Q
	#167 N0204chooseRegime:choosePumpRegime(start: #164, pump1Main: pin 18, pump2Main: pin 19, byCounter: #169, byWorkTime: pin 21)
	out 1 "выбран режим Н02.04/01 = главный" <= #167.pump1MainActive
	#168 N020402fTrigStop:F_TRIG(CLK: #170.pump2ON)
	out 2 "выбран режим Н02.04/02 = главный" <= #167.pump2MainActive
	out 3 "выбран режим по кол-ву включений" <= #167.byCounterActive
	#169 OR(pin 20, startInitializer)
	out 4 "выбран режим по наработке" <= #167.byWorkTimeActive
	#170 N0204manager:TwoPumpManager(startStopPump1: #167.startPump1, startStopPump2: #167.startPump2, alarmPump1: NOT pin 22, alarmPump2: NOT pin 23, alarmReset: pin 24, counterStart: #167.startByCounter, Pump1ResetCounter: pin 25, Pump2ResetCounter: pin 26, ValueToResetCounter: -, workTimeStart: #167.startByWorkTime, workTimePump1Reset: pin 27, workTimePump2Reset: pin 28)
	out 6 "пуск Н02.04/01" <= #170.pump1ON
	out 7 "пуск Н02.04/02" <= #170.pump2ON
	out 8 "счетчик включений Н02.04/01" <= #170.counterPump1
	out 9 "счетчик включений Н02.04/02" <= #170.counterPump2
	out 10 "счетчик наработки Н02.04/01" <= #170.currentWorkTimePump1
	out 11 "счетчик наработки Н02.04/02" <= #170.currentWorkTimePump2
END_MACRO
#171 N0204statRegimeP1M <= #158.out 1
#172 N0204statRegimeP2M <= #158.out 2
#173 N0204statRegimeByC <= #158.out 3
#174 N0204statRegimeWT <= #158.out 4
#175 DD4_DO.14 <= #158.out 5
#176 DD1_DO1 <= #158.out 6
#177 DD1_DO2 <= #158.out 7
#178 N0204counterP1 <= #158.out 8
#179 N0204counterP2 <= #158.out 9
#180 N0204workTimeP1 <= #158.out 10
#181 N0204workTimeP2 <= #158.out 11
#182 MACRO управление НД06.02 УПК(pin 1 "вход расходомера в куб/час": DD1_AI2_FT0102value, pin 2 "max производительность НД в мл/мин": ND0602setMaxDosVal, pin 3 "задание дозирования в мл/куб": ND0602setKoefProp, pin 4 "режим:1 насос главный": ND0602regimeP1M, pin 5 "режим: 2 насос главный": ND0602regimeP2M, pin 6 "режим: по наработке": ND0602regimeByWT, pin 7 "режим: по кол-ву включений": ND0602regimeByC, pin 8 "авария 1 насоса": DD6_DI.2, pin 9 "авария 2 насоса": DD6_DI.3, pin 10 "сброс аварий": alarmReset, pin 11 "сброс счетчика включений 1 насоса": ND0602resetCountP1, pin 12 "сброс ссчетчика включений 2 насоса": ND0602resetCountP2, pin 13 "сброс наработки 1 насоса": ND0602resetWorkTimeP1, pin 14 "сброс наработки 2 насоса": ND0602resetWorkTimeP2)
	(* Если на входе SEL = TRUE, / то нижнее значение, / иначе - то,что посередине. *)
	(* сигнал 4...20мА на НД06.02/01 *)
	(* сигнал 4...20мА на НД06.02/02 *)
	#183 SEL(#192.pump1ON, 4, #186.outputValue)
	#184 linTraf060201:LIN_TRAFO(IN: #183, IN_MIN: 4, IN_MAX: 20, OUT_MIN: 0, OUT_MAX: 1000)
	#185 REAL_TO_WORD(#184.OUT)
	out 6 "выход 4...20мА насоса 1" <= #185
	#186 ND0602dosing:DosingPumpProportional(flowValue: pin 1, setMinPumpDosingValue: -, setMaxPumpDosingValue: pin 2, minOutputValue: -, maxOutputValue: -, setKoeffProportionality: pin 3, minFlowToStart: -)
	out 1 "ошибка блока дозирования" <= #186.dosingError
	#187 SEL(#192.pump2ON, 4, #186.outputValue)
	#188 linTraf060202:LIN_TRAFO(IN: #187, IN_MIN: 4, IN_MAX: 20, OUT_MIN: 0, OUT_MAX: 1000)
	#189 REAL_TO_WORD(#188.OUT)
	out 7 "выход 4...20мА насоса 2" <= #189
	#190 ND0602regime:choosePumpRegime(start: #186.startDosingPump, pump1Main: pin 4, pump2Main: pin 5, byCounter: #191, byWorkTime: pin 6)
	out 2 "статус: 1 насос главный" <= #190.pump1MainActive
	out 3 "статус: 2 насос главный" <= #190.pump2MainActive
	out 4 "статус: по кол-ву включений" <= #190.byCounterActive
	#191 OR(pin 7, startInitializer)
	out 5 "статус: по наработке" <= #190.byWorkTimeActive
	#192 ND0602manager:TwoPumpManager(startStopPump1: #190.startPump1, startStopPump2: #190.startPump2, alarmPump1: #193, alarmPump2: #194, alarmReset: pin 10, counterStart: #190.startByCounter, Pump1ResetCounter: pin 11, Pump2ResetCounter: pin 12, ValueToResetCounter: -, workTimeStart: #190.startByWorkTime, workTimePump1Reset: pin 13, workTimePump2Reset: pin 14)
	out 12 "сигнал на включение насоса 1" <= #192.pump1ON
	#193 NOT(pin 8)
	out 13 "сигнал на включение насоса 2" <= #192.pump2ON
	out 8 "счетчик включений насоса 1" <= #192.counterPump1
	#194 NOT(pin 9)
	out 9 "счетчик включений насоса 2" <= #192.counterPump2
	out 10 "счетчик наработки насоса 1" <= #192.currentWorkTimePump1
	out 11 "счетчик наработки насоса 2" <= #192.currentWorkTimePump2
END_MACRO
#195 ND0602dosingError <= #182.out 1
#196 ND0602statRegimeP1M <= #182.out 2
#197 ND0602statRegimeP2M <= #182.out 3
#198 ND0602statRegimeByC <= #182.out 4
#199 ND0602statRegimeByWT <= #182.out 5
#200 DD10_AO1 <= #182.out 6
#201 DD10_AO2 <= #182.out 7
#202 ND0602counterP1 <= #182.out 8
#203 ND0602counterP2 <= #182.out 9
#204 ND0602workTimeP1 <= #182.out 10
#205 ND0602workTimeP2 <= #182.out 11
#206 DD4_DO.6 <= #182.out 12
#207 DD4_DO.7 <= #182.out 13
#208 OR(errorToOpenZDE0301, errorToCloseZDE0301, errorToOpenZDE0302, errorToCloseZDE0302)
#209 OR(DD5_DI.27, #208)
#210 OR(#208, DD5_DI.29)
#211 MACRO Работа УФО03.01(pin 1 "Работа УФО03.01/01": DD5_DI.26, pin 2 "Работа УФО03.01/02": DD5_DI.28, pin 3 "Значение расхода от FT01.02": DD1_AI2_FT0102value, pin 4 "мин.допустимый расход для насосов Н01.05": N0105minFlow, pin 5 "Задержка включения УФО на создание потока": UFO0301startDelayTime, pin 6 "выбор режим: УФО03.01/01 главное": UFO0301regimeP1M, pin 7 "выбор режим: УФО03.01/02 главное": UFO0301regimeP2M, pin 8 "выбор режим: по кол-ву включений": UFO0301regimeByC, pin 9 "выбор режим: по наработке": UFO0301regimeWT, pin 10 "авария УФО03.01/01": #209, pin 11 "авария УФО03.01/02": #210, pin 12 "сброс аварий": alarmReset, pin 13 "сброс счетчика включений УФО03.01/01": UFO0301resetCountP1, pin 14 "сброс счетчика включений УФО03.01/02": UFO0301resetCountP2, pin 15 "сброс счетчика наработки УФО03.01/01": UFO0301resetWorkTimeP1, pin 16 "сброс счетчика наработки УФО03.01/02": UFO0301resetWorkTimeP2)
	(* Включаем УФО, если расходомер показывает расход больше, / чем заданный как минимально допустимый для работы насосов Н01.05. *)
	(* Задержка старта УФО *)
	(* Для подачи предостережения на пульте / оператора (при необходимости), а также / сигнализации лампой АВАРИЯ. *)
	(* Контроль, если УФО включили вручную, / а потока при этом нет. *)
	#212 OR(pin 1, pin 2)
	#213 AND(#212, #214)
	out 1 "УФО вкл без потока" <= #213
	#214 NOT(#216.Q)
	#215 GE(pin 3, pin 4)
	#216 UFO0301startDelay:TON(IN: #215, PT: pin 5)
	#217 UFO0301regimeManager:choosePumpRegime(start: #216.Q, pump1Main: pin 6, pump2Main: pin 7, byCounter: #218, byWorkTime: pin 9)
	out 2 "активен режим - главное УФО 03.01/01" <= #217.pump1MainActive
	out 3 "активен режим - главное УФО 03.01/02" <= #217.pump2MainActive
	out 4 "активен режим - по кол-ву включений" <= #217.byCounterActive
	#218 OR(startInitializer, pin 8)
	out 5 "активен режим - по наработке" <= #217.byWorkTimeActive
	#219 UFO0301manager:TwoPumpManager(startStopPump1: #217.startPump1, startStopPump2: #217.startPump2, alarmPump1: pin 10, alarmPump2: pin 11, alarmReset: pin 12, counterStart: #217.startByCounter, Pump1ResetCounter: pin 13, Pump2ResetCounter: pin 14, ValueToResetCounter: -, workTimeStart: #217.startByWorkTime, workTimePump1Reset: pin 15, workTimePump2Reset: pin 16)
	out 6 "авт. пуск УФО03.01/01" <= #219.pump1ON
	out 7 "авт. пуск УФО03.01/02" <= #219.pump2ON
	out 8 "счетчик включений УФО03.01/01" <= #219.counterPump1
	out 9 "счетчик включений УФО03.01/02" <= #219.counterPump2
	out 10 "счетчик наработки УФО03.01/01" <= #219.currentWorkTimePump1
	out 11 "счетчик наработки УФО03.01/02" <= #219.currentWorkTimePump2
END_MACRO
#220 UFO0301noFlowAttention <= #211.out 1
#221 UFO0301statRegimeP1M <= #211.out 2
#222 UFO0301statRegimeP2M <= #211.out 3
#223 UFO0301statRegimeByC <= #211.out 4
#224 UFO0301statRegimeWT <= #211.out 5
#225 UFO0301counterP1 <= #211.out 8
#226 UFO0301counterP2 <= #211.out 9
#227 UFO0301workTimeP1 <= #211.out 10
#228 UFO0301workTimeP2 <= #211.out 11
#229 MACRO работа задвижек перед УФО и автом.пуск(pin 1 "сигнал на пуск УФО03.01/01": #211.out 6, pin 2 "сигнал на пуск УФО03.01/02": #211.out 7)
	(* 1 = открыть ЗДЭ03.02 / 0 = закрыть ЗДЭ03.02 *)
	(* 1 = открыть ЗДЭ03.01 / 0 = закрыть ЗДЭ03.01 *)
	(* 1 = тест задвижек ЗДЭ / 0 = возможность автом.пуска УФО *)
	(* авт.пускУФО03.01/01 *)
	(* авт.пускУФО03.01/02 *)
	#230 NOT(testZDE03)
	#231 NOT(testZDE03)
	#232 AND(#230, #234, DD1_DI12)
	#233 DD1_DO8 <= #232
	#234 SEL(testZDE03, pin 1, manualZDE0301)
	#235 ZDE0301:SimpleValve(inputOpen: #234, inputClose: NOT #234, statusOpen: DD1_DI12, statusClose: DD1_DI13, reset: alarmReset, timeToOpenClose: timeToOpenCloseValve)
	#236 DD4_DO.16 <= #235.outputOpen
	#237 DD4_DO.17 <= #235.outputClose
	#238 errorToOpenZDE0301 <= #235.errorToOpen
	#239 errorToCloseZDE0301 <= #235.errorToClose
	#240 AND(#231, #242, DD1_DI14)
	#241 DD1_DO9 <= #240
	#242 SEL(testZDE03, pin 2, manualZDE0302)
	#243 ZDE0302:SimpleValve(inputOpen: #242, inputClose: NOT #242, statusOpen: DD1_DI14, statusClose: DD1_DI15, reset: alarmReset, timeToOpenClose: timeToOpenCloseValve)
	#244 DD4_DO.18 <= #243.outputOpen
	#245 DD4_DO.19 <= #243.outputClose
	#246 errorToOpenZDE0302 <= #243.errorToOpen
	#247 errorToCloseZDE0302 <= #243.errorToClose
END_MACRO
#248 MACRO управление НД06.03 УПК(pin 1 "вход расходомера в куб/час": DD1_AI1_FT0101value, pin 2 "max производительность НД в мл/мин": ND0603setMaxDosVal, pin 3 "задание дозирования в мл/куб": ND0603setKoefProp, pin 4 "режим:1 насос главный": ND0603regimeP1M, pin 5 "режим: 2 насос главный": ND0603regimeP2M, pin 6 "режим: по наработке": ND0603regimeByWT, pin 7 "режим: по кол-ву включений": ND0603regimeByC, pin 8 "авария 1 насоса": DD6_DI.4, pin 9 "авария 2 насоса": DD6_DI.5, pin 10 "сброс аварий": alarmReset, pin 11 "сброс счетчика включений 1 насоса": ND0603resetCountP1, pin 12 "сброс ссчетчика включений 2 насоса": ND0603resetCountP2, pin 13 "сброс наработки 1 насоса": ND0603resetWorkTimeP1, pin 14 "сброс наработки 2 насоса": ND0603resetWorkTimeP2)
	(* Если на входе SEL = TRUE, / то нижнее значение, / иначе - то,что посередине. *)
	(* сигнал 4...20мА на НД06.03/01 *)
	(* сигнал 4...20мА на НД06.03/02 *)
	#249 SEL(#258.pump1ON, 4, #252.outputValue)
	#250 linTraf060301:LIN_TRAFO(IN: #249, IN_MIN: 4, IN_MAX: 20, OUT_MIN: 0, OUT_MAX: 1000)
	#251 REAL_TO_WORD(#250.OUT)
	out 6 "выход 4...20мА насоса 1" <= #251
	#252 ND0603dosing:DosingPumpProportional(flowValue: pin 1, setMinPumpDosingValue: -, setMaxPumpDosingValue: pin 2, minOutputValue: -, maxOutputValue: -, setKoeffProportionality: pin 3, minFlowToStart: -)
	out 1 "ошибка блока дозирования" <= #252.dosingError
	#253 SEL(#258.pump2ON, 4, #252.outputValue)
	#254 linTraf060302:LIN_TRAFO(IN: #253, IN_MIN: 4, IN_MAX: 20, OUT_MIN: 0, OUT_MAX: 1000)
	#255 REAL_TO_WORD(#254.OUT)
	out 7 "выход 4...20мА насоса 2" <= #255
	#256 ND0603regime:choosePumpRegime(start: #252.startDosingPump, pump1Main: pin 4, pump2Main: pin 5, byCounter: #257, byWorkTime: pin 6)
	out 2 "статус: 1 насос главный" <= #256.pump1MainActive
	out 3 "статус: 2 насос главный" <= #256.pump2MainActive
	out 4 "статус: по кол-ву включений" <= #256.byCounterActive
	#257 OR(pin 7, startInitializer)
	out 5 "статус: по наработке" <= #256.byWorkTimeActive
	#258 ND0603manager:TwoPumpManager(startStopPump1: #256.startPump1, startStopPump2: #256.startPump2, alarmPump1: #259, alarmPump2: #260, alarmReset: pin 10, counterStart: #256.startByCounter, Pump1ResetCounter: pin 11, Pump2ResetCounter: pin 12, ValueToResetCounter: -, workTimeStart: #256.startByWorkTime, workTimePump1Reset: pin 13, workTimePump2Reset: pin 14)
	out 12 "сигнал на включение насоса 1" <= #258.pump1ON
	#259 NOT(pin 8)
	out 13 "сигнал на включение насоса 2" <= #258.pump2ON
	out 8 "счетчик включений насоса 1" <= #258.counterPump1
	#260 NOT(pin 9)
	out 9 "счетчик включений насоса 2" <= #258.counterPump2
	out 10 "счетчик наработки насоса 1" <= #258.currentWorkTimePump1
	out 11 "счетчик наработки насоса 2" <= #258.currentWorkTimePump2
END_MACRO
#261 ND0603dosingError <= #248.out 1
#262 ND0603statRegimeP1M <= #248.out 2
#263 ND0603statRegimeP2M <= #248.out 3
#264 ND0603statRegimeByC <= #248.out 4
#265 ND0603statRegimeByWT <= #248.out 5
#266 DD10_AO3 <= #248.out 6
#267 DD10_AO4 <= #248.out 7
#268 ND0603counterP1 <= #248.out 8
#269 ND0603counterP2 <= #248.out 9
#270 ND0603workTimeP1 <= #248.out 10
#271 ND0603workTimeP2 <= #248.out 11
#272 DD4_DO.8 <= #248.out 12
#273 DD4_DO.9 <= #248.out 13
#274 MACRO управление Н04.04 (дренажные)(pin 1 "защита от сухого хода Н04.04": DD5_DI.18, pin 2 "автоматич.пускН04.04": DD5_DI.19, pin 3 "режим Н04.04/01 главный": N0404regimeP1M, pin 4 "режим Н04.04/02 главный": N0404regimeP2M, pin 5 "режим по кол-ву включений": N0404regimeByC, pin 6 "режим по наработке": N0404regimeWT, pin 7 "авария Н04.04/01": DD5_DI.15, pin 8 "авария Н04.04/02": DD5_DI.14, pin 9 "сброс аварий": alarmReset, pin 10 "сброс счетчика включений Н04.04/01": N0404resetCountP1, pin 11 "сброс счетчика включений Н04.04/02": N0404resetCountP2, pin 12 "сброс счетчика наработки Н04.04/01": N0404resetWorkTimeP1, pin 13 "сброс счетчика наработки Н04.04/02": N0404resetWorkTimeP2)
	(* 0=авария *)
	(* сухой ход Н04.04 / 0=защита *)
	(* от поплавка *)
	(* насосы имеют электрическую блокировку / от одновременного включения *)
	(* Излишняя перестраховка по сухому ходу, / на уровне реле уже все отрабатывается. *)
	(* сбрасывает самоподхват пускового реле *)
	#275 NOT(pin 1)
	out 1 "стоп Н04.04" <= #275
	#276 AND(pin 1, pin 2)
	#277 N0401choosePumpRegime:choosePumpRegime(start: #276, pump1Main: pin 3, pump2Main: pin 4, byCounter: #278, byWorkTime: pin 6)
	out 2 "выбран режим: Н04.04/01 главный" <= #277.pump1MainActive
	out 3 "выбран режим: Н04.04/02 главный" <= #277.pump2MainActive
	out 4 "выбран режим: по кол-ву включений" <= #277.byCounterActive
	#278 OR(startInitializer, pin 5)
	out 5 "выбран режим: по наработке" <= #277.byWorkTimeActive
	#279 N0404twoPumpManager:TwoPumpManager(startStopPump1: #277.startPump1, startStopPump2: #277.startPump2, alarmPump1: #280, alarmPump2: #281, alarmReset: pin 9, counterStart: #277.startByCounter, Pump1ResetCounter: pin 10, Pump2ResetCounter: pin 11, ValueToResetCounter: -, workTimeStart: #277.startByWorkTime, workTimePump1Reset: pin 12, workTimePump2Reset: pin 13)
	out 6 "пуск Н04.04/01" <= #279.pump1ON
	#280 NOT(pin 7)
	out 7 "пуск Н04.04/02" <= #279.pump2ON
	out 8 "счетчик кол-ва включений Н04.04/01" <= #279.counterPump1
	#281 NOT(pin 8)
	out 9 "счетчик кол-ва включений Н04.04/02" <= #279.counterPump2
	out 10 "счетчик времени наработки Н04.04/01" <= #279.currentWorkTimePump1
	out 11 "счетчик времени наработки Н04.04/02" <= #279.currentWorkTimePump2
END_MACRO
#282 DD4_DO.15 <= #274.out 1
#283 N0404statRegimeP1M <= #274.out 2
#284 N0404statRegimeP2M <= #274.out 3
#285 N0404statRegimeByC <= #274.out 4
#286 N0404statRegimeWT <= #274.out 5
#287 DD1_DO5 <= #274.out 6
#288 DD1_DO6 <= #274.out 7
#289 N0404counterP1 <= #274.out 8
#290 N0404counterP2 <= #274.out 9
#291 N0404workTimeP1 <= #274.out 10
#292 N0404workTimeP2 <= #274.out 11
#293 MACRO управление НД07.03 УПЩ (поддержка рН, ПИД-регулятор)(pin 1 "вход рН-метра QE01.01": DD1_AI3_QE0101value, pin 2 "уставка рН": ND0703pHsetValue, pin 3 "режим:1 насос главный": ND0703regimeP1M, pin 4 "режим: 2 насос главный": ND0703regimeP2M, pin 5 "режим: по наработке": ND0703regimeByWT, pin 6 "режим: по кол-ву включений": ND0703regimeByC, pin 7 "авария 1 насоса": DD6_DI.6, pin 8 "авария 2 насоса": DD6_DI.7, pin 9 "сброс аварий": alarmReset, pin 10 "сброс счетчика включений 1 насоса": ND0703resetCountP1, pin 11 "сброс счетчика включений 2 насоса": ND0703resetCountP2, pin 12 "сброс наработки 1 насоса": ND0703resetWorkTimeP1, pin 13 "сброс наработки 2 насоса": ND0703resetWorkTimeP2, pin 14 "ручное управл.выходом Y (4...20мА)": ND0703YoutManual, pin 15 "1=ручное/0=автомат.управл.": ND0703YmanAuto, pin 16 "вход расходомера FT01.01 (куб.м/час)": DD1_AI1_FT0101value, pin 17 "коэфф.I": ND0703koeffI, pin 18 "коэфф.D": ND0703koeffD, pin 19 "коэфф.Р": ND0703koeffP)
	(* min расход в кубометрах в час / для неачала дозирования. *)
	(* Если на входе SEL = TRUE, / то нижнее значение, / иначе - то,что посередине. *)
	(* сигнал 4...20мА на НД07.03/01 *)
	(* сигнал 4...20мА на НД07.03/02 *)
	#294 ND0703pidReg:PID(ACTUAL: pin 1, SET_POINT: pin 2, KP: pin 19, TN: pin 17, TV: pin 18, Y_MANUAL: pin 14, Y_OFFSET: 500, Y_MIN: 0, Y_MAX: 1000, MANUAL: pin 15, RESET: #294.OVERFLOW)
	#295 SEL(#302.pump1ON, 0, #294.Y)
	#296 REAL_TO_WORD(#295)
	out 5 "выход 4...20мА насоса 1" <= #296
	#297 SEL(#302.pump2ON, 0, #294.Y)
	#298 REAL_TO_WORD(#297)
	out 6 "выход 4...20мА насоса 2" <= #298
	#299 GE(pin 16, 10)
	#300 ND0703regime:choosePumpRegime(start: #299, pump1Main: pin 3, pump2Main: pin 4, byCounter: #301, byWorkTime: pin 5)
	out 1 "статус: 1 насос главный" <= #300.pump1MainActive
	out 2 "статус: 2 насос главный" <= #300.pump2MainActive
	out 3 "статус: по кол-ву включений" <= #300.byCounterActive
	out 4 "статус: по наработке" <= #300.byWorkTimeActive
	#301 OR(pin 6, startInitializer)
	#302 ND0703manager:TwoPumpManager(startStopPump1: #300.startPump1, startStopPump2: #300.startPump2, alarmPump1: #303, alarmPump2: #304, alarmReset: pin 9, counterStart: #300.startByCounter, Pump1ResetCounter: pin 10, Pump2ResetCounter: pin 11, ValueToResetCounter: -, workTimeStart: #300.startByWorkTime, workTimePump1Reset: pin 12, workTimePump2Reset: pin 13)
	out 11 "сигнал на включение насоса 1" <= #302.pump1ON
	#303 NOT(pin 7)
	out 12 "сигнал на включение насоса 2" <= #302.pump2ON
	out 7 "счетчик включений насоса 1" <= #302.counterPump1
	#304 NOT(pin 8)
	out 8 "счетчик включений насоса 2" <= #302.counterPump2
	out 9 "счетчик наработки насоса 1" <= #302.currentWorkTimePump1
	out 10 "счетчик наработки насоса 2" <= #302.currentWorkTimePump2
END_MACRO
#305 ND0703statRegimeP1M <= #293.out 1
#306 ND0703statRegimeP2M <= #293.out 2
#307 ND0703statRegimeByC <= #293.out 3
#308 ND0703statRegimeByWT <= #293.out 4
#309 DD10_AO5 <= #293.out 5
#310 DD10_AO6 <= #293.out 6
#311 ND0703counterP1 <= #293.out 7
#312 ND0703counterP2 <= #293.out 8
#313 ND0703workTimeP1 <= #293.out 9
#314 ND0703workTimeP2 <= #293.out 10
#315 DD4_DO.10 <= #293.out 11
#316 DD4_DO.11 <= #293.out 12
#317 MACRO импульсный счетчик FQS0301(pin 1 "вход от счетчика": DD6_DI.19, pin 2 "вес импульса счетчика": FQS0301impulsValue, pin 3 "сброс счетчика": FQS0301reset, pin 4 "величина коррекции счетчика": FQS0301correction, pin 5 "прибавить коррекцию": FQS0301addCorrection, pin 6 "вычесть коррекцию": FQS0301deleteCorrection)
	(* число, коорое будем прибавлять или / вычитать из накопленной суммы стоков. *)
	(* коррекция показаний счетчика. *)
	(* Если в результате коррекции накопленная сумма станет меньше нуля, то она принудительно станет равна нулю. *)
	(* значение в REAL (в какой-то момент начинает / отображаться в экспоненциальной форме) *)
	(* сброс показаний счетчика *)
	#318 FQS0301rTrig:R_TRIG(CLK: pin 1)
	#319 ADD(EN: #318.Q, FQS0301totalAmount, pin 2)
	out 1 "накопленная сумма стоков (REAL)" <= #319
	#320 FQS0301resetRtrig:R_TRIG(CLK: pin 3)
	#321 MOVE(EN: #320.Q, 0)
	#322 FQS0301totalAmount <= #321
	#323 FQS0301addCorrRtrig:R_TRIG(CLK: pin 5)
	#324 ADD(EN: #323.Q, FQS0301totalAmount, pin 4)
	#325 FQS0301totalAmount <= #324
	#326 FQS0301deleteCorrRtrig:R_TRIG(CLK: pin 6)
	#327 SUB(EN: #326.Q, FQS0301totalAmount, pin 4)
	#328 FQS0301totalAmount <= #327
	#329 LT(FQS0301totalAmount, 0)
	#330 MOVE(EN: #329, 0)
	#331 FQS0301totalAmount <= #330
END_MACRO
#332 FQS0301totalAmount <= #317.out 1
#333 MACRO управление НД08.03 УПФ(pin 1 "вход расходомера в куб/час": DD1_AI1_FT0101value, pin 2 "max производительность НД в мл/мин": ND0803setMaxDosVal, pin 3 "задание дозирования в мл/куб": ND0803setKoefProp, pin 4 "режим:1 насос главный": ND0803regimeP1M, pin 5 "режим: 2 насос главный": ND0803regimeP2M, pin 6 "режим: по наработке": ND0803regimeByWT, pin 7 "режим: по кол-ву включений": ND0803regimeByC, pin 8 "авария 1 насоса": DD5_DI.12, pin 9 "авария 2 насоса": DD5_DI.13, pin 10 "сброс аварий": alarmReset, pin 11 "сброс счетчика включений 1 насоса": ND0803resetCountP1, pin 12 "сброс ссчетчика включений 2 насоса": ND0803resetCountP2, pin 13 "сброс наработки 1 насоса": ND0803resetWorkTimeP1, pin 14 "сброс наработки 2 насоса": ND0803resetWorkTimeP2, pin 15 "сухой ход 1 насоса": DD1_DI6, pin 16 "сухой ход 2 насоса": DD1_DI7)
	(* Если на входе SEL = TRUE, / то нижнее значение, / иначе - то,что посередине. *)
	(* сигнал 4...20мА на НД08.03/01 *)
	(* сигнал 4...20мА на НД08.03/02 *)
	#334 SEL(#343.pump1ON, 0, #335.outputValue)
	out 6 "выход 4...20мА насоса 1" <= #334
	#335 ND0803dosing:DosingPumpProportional(flowValue: pin 1, setMinPumpDosingValue: -, setMaxPumpDosingValue: pin 2, minOutputValue: -, maxOutputValue: -, setKoeffProportionality: pin 3, minFlowToStart: -)
	out 1 "ошибка блока дозирования" <= #335.dosingError
	#336 SEL(#343.pump2ON, 0, #335.outputValue)
	out 7 "выход 4...20мА насоса 2" <= #336
	#337 ND0803regime:choosePumpRegime(start: #335.startDosingPump, pump1Main: pin 4, pump2Main: pin 5, byCounter: #338, byWorkTime: pin 6)
	out 2 "статус: 1 насос главный" <= #337.pump1MainActive
	out 3 "статус: 2 насос главный" <= #337.pump2MainActive
	out 4 "статус: по кол-ву включений" <= #337.byCounterActive
	#338 OR(pin 7, startInitializer)
	out 5 "статус: по наработке" <= #337.byWorkTimeActive
	out 12 "сигнал на включение насоса 1" <= #343.pump1ON
	#339 NOT(pin 8)
	#340 OR(#339, pin 15)
	out 13 "сигнал на включение насоса 2" <= #343.pump2ON
	#341 NOT(pin 9)
	#342 OR(#341, pin 16)
	#343 ND0803manager:TwoPumpManager(startStopPump1: #337.startPump1, startStopPump2: #337.startPump2, alarmPump1: #340, alarmPump2: #342, alarmReset: pin 10, counterStart: #337.startByCounter, Pump1ResetCounter: pin 11, Pump2ResetCounter: pin 12, ValueToResetCounter: -, workTimeStart: #337.startByWorkTime, workTimePump1Reset: pin 13, workTimePump2Reset: pin 14)
	out 8 "счетчик включений насоса 1" <= #343.counterPump1
	out 9 "счетчик включений насоса 2" <= #343.counterPump2
	out 10 "счетчик наработки насоса 1" <= #343.currentWorkTimePump1
	out 11 "счетчик наработки насоса 2" <= #343.currentWorkTimePump2
END_MACRO
#344 ND0803dosingError <= #333.out 1
#345 ND0803statRegimeP1M <= #333.out 2
#346 ND0803statRegimeP2M <= #333.out 3
#347 ND0803statRegimeByC <= #333.out 4
#348 ND0803statRegimeByWT <= #333.out 5
#349 DD1_AO1 <= #333.out 6
#350 DD1_AO2 <= #333.out 7
#351 ND0803counterP1 <= #333.out 8
#352 ND0803counterP2 <= #333.out 9
#353 ND0803workTimeP1 <= #333.out 10
#354 ND0803workTimeP2 <= #333.out 11
#355 DD1_DO3 <= #333.out 12
#356 DD1_DO4 <= #333.out 13
#357 AND(DD1_DI5, DD1_DI4, DD6_DI.11)
#358 DD1_DO8 <= #357
#359 EQ(lastError, 0)
#360 alarmPLKnetworkDelay:TOF(IN: #359, PT: T#20s)
#361 NOT(#360.Q)
#362 alarmPLKnetwork <= #361
#363 MACRO управление НД08.04 УПФ(pin 1 "насос Н04.01 работает": DD7_DI.13, pin 2 "авария НД08.04": DD6_DI.16, pin 3 "уставкаНД08.04(0...100%)": ND0804doseValue)
	(* Преобразует сигнал 0...100 / пропорционально в 4...20мА, / в модуль АО подаем 0...1000. *)
	#364 AND(pin 1, pin 2)
	out 1 "пуск/стоп НД08.04" <= #364
	#365 ND0804linearTransformator:LIN_TRAFO(IN: pin 3, IN_MIN: 0, IN_MAX: 100, OUT_MIN: 0, OUT_MAX: 1000)
	#366 REAL_TO_WORD(#365.OUT)
	out 2 "управление НД08.04 (4...20мА)" <= #366
	out 3 "ошибка блока дозирования" <= #365.ERROR
END_MACRO
#367 DD4_DO.12 <= #363.out 1
#368 DD10_AO7 <= #363.out 2
#369 ND0804dosingError <= #363.out 3
#370 NOT(DD6_DI.0)
#371 alarmND050201 <= #370
#372 NOT(DD6_DI.23)
#373 alarmFS020102 <= #372
#374 NOT(DD9_DI.14)
#375 alarmZDE0211power <= #374
#376 NOT(DD6_DI.1)
#377 alarmND050202 <= #376
#378 NOT(DD6_DI.25)
#379 alarmFS020103 <= #378
#380 NOT(DD9_DI.15)
#381 alarmZDE0212power <= #380
#382 NOT(DD6_DI.2)
#383 alarmND060201 <= #382
#384 NOT(DD6_DI.27)
#385 alarmFS020104 <= #384
#386 NOT(DD9_DI.16)
#387 alarmZDE0213power <= #386
#388 NOT(DD6_DI.3)
#389 alarmND060202 <= #388
#390 NOT(DD6_DI.29)
#391 alarmFS020105 <= #390
#392 NOT(DD9_DI.17)
#393 alarmZDE0214power <= #392
#394 MACRO контроль включения мешалок(pin 1 "работа НД06.02/01": DD4_DO.6, pin 2 "работа НД06.02/02": DD4_DO.7, pin 3 "работа НД06.03/01": DD4_DO.8, pin 4 "работа НД06.03/02": DD4_DO.9, pin 5 "работа мешалки М06.04": DD5_DI.21, pin 6 "работа НД07.03/01": DD4_DO.10, pin 7 "работа НД07.03/02": DD4_DO.11, pin 8 "работа мешалки М07.02": DD5_DI.23, pin 9 "работа НД08.03/01": DD1_DO3, pin 10 "работа НД08.03/02": DD1_DO4, pin 11 "работа НД08.04": DD4_DO.12, pin 12 "работа мешалки М08.02": DD5_DI.25)
	#395 OR(pin 1, pin 2, pin 3, pin 4)
	#396 AND(#395, #397)
	out 1 "дозирования при выключенной М06.04" <= #396
	#397 NOT(pin 5)
	#398 OR(pin 6, pin 7)
	#399 AND(#398, #400)
	out 2 "дозирования при выключенной М07.02" <= #399
	#400 NOT(pin 8)
	#401 OR(pin 9, pin 10, pin 11)
	#402 AND(#401, #403)
	out 3 "дозирования при выключенной М08.02" <= #402
	#403 NOT(pin 12)
END_MACRO
#404 M0604attention <= #394.out 1
#405 M0702attention <= #394.out 2
#406 M0802attention <= #394.out 3
#407 NOT(DD6_DI.4)
#408 alarmND060301 <= #407
#409 NOT(DD6_DI.31)
#410 alarmFS020106 <= #409
#411 NOT(DD9_DI.18)
#412 alarmZDE0215power <= #411
#413 NOT(DD6_DI.5)
#414 alarmND060302 <= #413
#415 NOT(DD7_DI.1)
#416 alarmFS020201 <= #415
#417 NOT(DD9_DI.19)
#418 alarmZDE0216power <= #417
#419 NOT(DD6_DI.6)
#420 alarmND070301 <= #419
#421 NOT(DD7_DI.3)
#422 alarmFS020202 <= #421
#423 NOT(DD9_DI.20)
#424 alarmZDE0217power <= #423
#425 NOT(DD6_DI.7)
#426 alarmND070302 <= #425
#427 NOT(DD7_DI.5)
#428 alarmFS020203 <= #427
#429 NOT(DD9_DI.21)
#430 alarmZDE0218power <= #429
#431 NOT(DD5_DI.12)
#432 alarmND080301 <= #431
#433 NOT(DD7_DI.7)
#434 alarmFS020204 <= #433
#435 NOT(DD9_DI.22)
#436 alarmZDE0219power <= #435
#437 NOT(DD5_DI.13)
#438 alarmND080302 <= #437
#439 NOT(DD7_DI.9)
#440 alarmFS020205 <= #439
#441 NOT(DD9_DI.23)
#442 alarmZDE0220power <= #441
#443 NOT(DD6_DI.16)
#444 alarmND0804 <= #443
#445 NOT(DD7_DI.11)
#446 alarmFS020206 <= #445
#447 NOT(DD9_DI.24)
#448 alarmZDE0221power <= #447
#449 NOT(DD6_DI.11)
#450 alarmOGM0104overload <= #449
#451 NOT(DD9_DI.4)
#452 alarmZDE0201power <= #451
#453 NOT(DD9_DI.25)
#454 alarmZDE0222power <= #453
#455 MACRO переменные для обмена с панелью()
	#456 MACRO PSW регистры на передачу в панель (отображение)()
		(* panFQS0301totalAmount - переменная отображена сразу на выходе соответствующего макроса (учет очищенных стоков). / Здесь не хранится. *)
		(* PSW регистры на передачу в панель (отображение) *)
		#457 panFT0101value <= DD1_AI1_FT0101value
		#458 panQE0101value <= DD1_AI3_QE0101value
		#459 panFT0102value <= DD1_AI2_FT0102value
		#460 panQE0102value <= DD1_AI4_QE0102value
		#461 panFPKpressureValue <= DD1_AI5_FPKpressureValue
		#462 panFQS0301total <= FQS0301totalAmount
		#463 panTemperature <= temperatureValue
		#464 MACRO Время наработки и кол-во включений агрегатов()
			#465 workTimeND050201:TimeFromWorkTime(input: ND0502workTimeP1)
			#466 panND050201workDays <= #465.days
			#467 panND050201workHours <= #465.hours
			#468 panND050201workMinutes <= #465.minutes
			#469 panND050201workSeconds <= #465.seconds
			#470 workTimeND050202:TimeFromWorkTime(input: ND0502workTimeP2)
			#471 panND050202workDays <= #470.days
			#472 panND050202workHours <= #470.hours
			#473 panND050202workMinutes <= #470.minutes
			#474 panND050202workSeconds <= #470.seconds
			#475 panND0502counterP1 <= ND0502counterP1
			#476 panND0502counterP2 <= ND0502counterP2
			#477 workTimeND060201:TimeFromWorkTime(input: ND0602workTimeP1)
			#478 panND060201workDays <= #477.days
			#479 panND060201workHours <= #477.hours
			#480 panND060201workMinutes <= #477.minutes
			#481 panND060201workSeconds <= #477.seconds
			#482 workTimeND060202:TimeFromWorkTime(input: ND0602workTimeP2)
			#483 panND060202workDays <= #482.days
			#484 panND060202workHours <= #482.hours
			#485 panND060202workMinutes <= #482.minutes
			#486 panND060202workSeconds <= #482.seconds
			#487 panND0602counterP1 <= ND0602counterP1
			#488 panND0602counterP2 <= ND0602counterP2
			#489 workTimeND060301:TimeFromWorkTime(input: ND0603workTimeP1)
			#490 panND060301workDays <= #489.days
			#491 panND060301workHours <= #489.hours
			#492 panND060301workMinutes <= #489.minutes
			#493 panND060301workSeconds <= #489.seconds
			#494 workTimeND060302:TimeFromWorkTime(input: ND0603workTimeP2)
			#495 panND060302workDays <= #494.days
			#496 panND060302workHours <= #494.hours
			#497 panND060302workMinutes <= #494.minutes
			#498 panND060302workSeconds <= #494.seconds
			#499 panND0603counterP1 <= ND0603counterP1
			#500 panND0603counterP2 <= ND0603counterP2
			#501 workTimeND070301:TimeFromWorkTime(input: ND0703workTimeP1)
			#502 panND070301workDays <= #501.days
			#503 panND070301workHours <= #501.hours
			#504 panND070301workMinutes <= #501.minutes
			#505 panND070301workSeconds <= #501.seconds
			#506 workTimeND070302:TimeFromWorkTime(input: ND0703workTimeP2)
			#507 panND070302workDays <= #506.days
			#508 panND070302workHours <= #506.hours
			#509 panND070302workMinutes <= #506.minutes
			#510 panND070302workSeconds <= #506.seconds
			#511 panND0703counterP1 <= ND0703counterP1
			#512 panND0703counterP2 <= ND0703counterP2
			#513 workTimeND080301:TimeFromWorkTime(input: ND0803workTimeP1)
			#514 panND080301workDays <= #513.days
			#515 panND080301workHours <= #513.hours
			#516 panND080301workMinutes <= #513.minutes
			#517 panND080301workSeconds <= #513.seconds
			#518 workTimeND080302:TimeFromWorkTime(input: ND0803workTimeP2)
			#519 panND080302workDays <= #518.days
			#520 panND080302workHours <= #518.hours
			#521 panND080302workMinutes <= #518.minutes
			#522 panND080302workSeconds <= #518.seconds
			#523 panND0803counterP1 <= ND0803counterP1
			#524 panND0803counterP2 <= ND0803counterP2
			#525 workTimeN010501:TimeFromWorkTime(input: N0105workTimeP1)
			#526 panN010501workDays <= #525.days
			#527 panN010501workHours <= #525.hours
			#528 panN010501workMinutes <= #525.minutes
			#529 panN010501workSeconds <= #525.seconds
			#530 workTimeN010502:TimeFromWorkTime(input: N0105workTimeP2)
			#531 panN010502workDays <= #530.days
			#532 panN010502workHours <= #530.hours
			#533 panN010502workMinutes <= #530.minutes
			#534 panN010502workSeconds <= #530.seconds
			#535 panN0105counterP1 <= N0105counterP1
			#536 panN0105counterP2 <= N0105counterP2
			#537 workTimeN020401:TimeFromWorkTime(input: N0204workTimeP1)
			#538 panN020401workDays <= #537.days
			#539 panN020401workHours <= #537.hours
			#540 panN020401workMinutes <= #537.minutes
			#541 panN020401workSeconds <= #537.seconds
			#542 workTimeN020402:TimeFromWorkTime(input: N0204workTimeP2)
			#543 panN020402workDays <= #542.days
			#544 panN020402workHours <= #542.hours
			#545 panN020402workMinutes <= #542.minutes
			#546 panN020402workSeconds <= #542.seconds
			#547 panN0204counterP1 <= N0204counterP1
			#548 panN0204counterP2 <= N0204counterP2
			#549 workTimeN040401:TimeFromWorkTime(input: N0404workTimeP1)
			#550 panN040401workDays <= #549.days
			#551 panN040401workHours <= #549.hours
			#552 panN040401workMinutes <= #549.minutes
			#553 panN040401workSeconds <= #549.seconds
			#554 workTimeN040402:TimeFromWorkTime(input: N0404workTimeP2)
			#555 panN040402workDays <= #554.days
			#556 panN040402workHours <= #554.hours
			#557 panN040402workMinutes <= #554.minutes
			#558 panN040402workSeconds <= #554.seconds
			#559 panN0404counterP1 <= N0404counterP1
			#560 panN0404counterP2 <= N0404counterP2
			#561 workTimeUFO030101:TimeFromWorkTime(input: UFO0301workTimeP1)
			#562 panUFO030101workDays <= #561.days
			#563 panUFO030101workHours <= #561.hours
			#564 panUFO030101workMinutes <= #561.minutes
			#565 panUFO030101workSeconds <= #561.seconds
			#566 workTimeUFO030102:TimeFromWorkTime(input: UFO0301workTimeP2)
			#567 panUFO030102workDays <= #566.days
			#568 panUFO030102workHours <= #566.hours
			#569 panUFO030102workMinutes <= #566.minutes
			#570 panUFO030102workSeconds <= #566.seconds
			#571 panUFO0301counterP1 <= UFO0301counterP1
			#572 panUFO0301counterP2 <= UFO0301counterP2
		END_MACRO
	END_MACRO
	#573 MACRO PSB регистры на передачу в панель (отображение)()
		(* PSB регистры на передачу в панель (отображение) *)
		#574 MACRO 8 bit output module 1()
			#575 panStartND050201 <= DD4_DO.4
			#576 panStartND050202 <= DD4_DO.5
			#577 panStartND060201 <= DD4_DO.6
			#578 panStartND060202 <= DD4_DO.7
			#579 panStartND060301 <= DD4_DO.8
			#580 panStartND060302 <= DD4_DO.9
			#581 panStartM0604 <= DD5_DI.21
			#582 panStartND070301 <= DD4_DO.10
		END_MACRO
		#583 MACRO 8 bit output module 2()
			#584 panStartND070302 <= DD4_DO.11
			#585 panStartM0702 <= DD5_DI.23
			#586 panStartND080301 <= DD1_DO3
			#587 panStartND080302 <= DD1_DO4
			#588 panStartND0804 <= DD4_DO.12
			#589 panStartM0802 <= DD5_DI.25
			#590 panStartN020401 <= DD5_DI.9
			#591 panStartN020402 <= DD5_DI.10
		END_MACRO
		#592 MACRO 8 bit output module 3()
			#593 panStartN010501 <= N0105statStartedP1
			#594 panStartN010502 <= N0105statStartedP2
			#595 panCleanFS020101 <= DD6_DI.20
			#596 panCleanFS020102 <= DD6_DI.22
			#597 panCleanFS020103 <= DD6_DI.24
			#598 panCleanFS020104 <= DD6_DI.26
			#599 panCleanFS020105 <= DD6_DI.28
			#600 panCleanFS020106 <= DD6_DI.30
		END_MACRO
		#601 MACRO 8 bit output module 4()
			#602 panCleanFS020201 <= DD7_DI. 0
			#603 panCleanFS020202 <= DD7_DI. 2
			#604 panCleanFS020203 <= DD7_DI. 4
			#605 panCleanFS020204 <= DD7_DI. 6
			#606 panCleanFS020205 <= DD7_DI. 8
			#607 panCleanFS020206 <= DD7_DI. 10
			#608 panSludgeReady <= DD7_DI.15
			#609 panStartN0401 <= DD7_DI.13
		END_MACRO
		#610 MACRO 8 bit output module 5()
			#611 panKSHE0401open <= DD9_DI.2
			#612 panFPKready <= DD7_DI.12
			#613 panFPKneedToClean <= FPKneedToClean
			#614 panStartN040401 <= DD5_DI.16
			#615 panStartN040402 <= DD5_DI.17
			#616 panStartUFO030101 <= DD5_DI.26
			#617 panStartUFO030102 <= DD5_DI.28
			#618 panAlarm <= alarm
		END_MACRO
		#619 MACRO 8 bit output module 6()
			#620 panErrorTempSensor <= DD1_AI0_error
			#621 panErrorFT0101 <= DD1_AI1_error
			#622 panErrorFT0102 <= DD1_AI2_error
			#623 panErrorQE0102 <= DD1_AI3_error
			#624 panErrorQE0102 <= DD1_AI4_error
			#625 panAlarmHighTemp <= alarmHighTemperature
			#626 panAlarmLowTemp <= alarmLowTemperature
			#627 panND0502dosingError <= ND0502dosingError
		END_MACRO
		#628 MACRO 8 bit output module 7()
			#629 panND0602dosingError <= ND0602dosingError
			#630 panND0603dosingError <= ND0603dosingError
			#631 panND0803dosingError <= ND0803dosingError
			#632 panND0804dosingError <= ND0804dosingError
			#633 panND080301emptyAlarm <= DD1_DI6
			#634 panND080302emptyAlarm <= DD1_DI7
			#635 panN010501alarm <= N010501alarm
			#636 panN010502alarm <= N010502alarm
		END_MACRO
		#637 MACRO 8 bit output module 8()
			#638 panZDE0225errorToOpen <= ZDE0225errorToOpen
			#639 panZDE0225errorToClose <= ZDE0225errorToClose
			#640 panFPKalarm <= DD7_DI.14
			#641 panFPKnotStarted <= FPKnotStarted
			#642 panErrorFPKsensor <= DD1_AI5_error
			#643 panFPKkshe0401errorToOpen <= FPKkshe0401errorToOpen
			#644 panFPKkshe0401errorToClose <= FPKkshe0401errorToClose
			#645 panUFO030101alarm <= DD5_DI.27
		END_MACRO
		#646 MACRO 8 bit output module 9()
			#647 panUFO030102alarm <= DD5_DI.29
			#648 panFilterFailToRegen020101 <= filterFailToRegen020101
			#649 panErrorToOpenZD0201 <= errorToOpenZD0201
			#650 panErrorToCloseZD0201 <= errorToCloseZD0201
			#651 panErrorToOpenZD0207 <= errorToOpenZD0207
			#652 panErrorToCloseZD0207 <= errorToCloseZD0207
			#653 panFilterFailToRegen020102 <= filterFailToRegen020102
			#654 panErrorToOpenZD0202 <= errorToOpenZD0202
		END_MACRO
		#655 MACRO 8 bit output module 10()
			#656 panErrorToCloseZD0202 <= errorToCloseZD0202
			#657 panErrorToOpenZD0208 <= errorToOpenZD0208
			#658 panErrorToCloseZD0208 <= errorToCloseZD0208
			#659 panFilterFailToRegen020103 <= filterFailToRegen020103
			#660 panErrorToOpenZD0203 <= errorToOpenZD0203
			#661 panErrorToCloseZD0203 <= errorToCloseZD0203
			#662 panErrorToOpenZD0209 <= errorToOpenZD0209
			#663 panErrorToCloseZD0209 <= errorToCloseZD0209
		END_MACRO
		#664 MACRO 8 bit output module 11()
			#665 panFilterFailToRegen020104 <= filterFailToRegen020104
			#666 panErrorToOpenZD0204 <= errorToOpenZD0204
			#667 panErrorToCloseZD0204 <= errorToCloseZD0204
			#668 panErrorToOpenZD0210 <= errorToOpenZD0210
			#669 panErrorToCloseZD0210 <= errorToCloseZD0210
			#670 panFilterFailToRegen020105 <= filterFailToRegen020105
			#671 panErrorToOpenZD0205 <= errorToOpenZD0205
			#672 panErrorToCloseZD0205 <= errorToCloseZD0205
		END_MACRO
		#673 MACRO 8 bit output module 12()
			#674 panErrorToOpenZD0211 <= errorToOpenZD0211
			#675 panErrorToCloseZD0211 <= errorToCloseZD0211
			#676 panFilterFailToRegen020106 <= filterFailToRegen020106
			#677 panErrorToOpenZD0206 <= errorToOpenZD0206
			#678 panErrorToCloseZD0206 <= errorToCloseZD0206
			#679 panErrorToOpenZD0212 <= errorToOpenZD0212
			#680 panErrorToCloseZD0212 <= errorToCloseZD0212
			#681 panFilterFailToRegen020201 <= filterFailToRegen020201
		END_MACRO
		#682 MACRO 8 bit output module 13()
			#683 panErrorToOpenZD0213 <= errorToOpenZD0213
			#684 panErrorToCloseZD0213 <= errorToCloseZD0213
			#685 panErrorToOpenZD0219 <= errorToOpenZD0219
			#686 panErrorToCloseZD0219 <= errorToCloseZD0219
			#687 panFilterFailToRegen020202 <= filterFailToRegen020202
			#688 panErrorToOpenZD0214 <= errorToOpenZD0214
			#689 panErrorToCloseZD0214 <= errorToCloseZD0214
			#690 panErrorToOpenZD0220 <= errorToOpenZD0220
		END_MACRO
		#691 MACRO 8 bit output module 14()
			#692 panErrorToCloseZD0220 <= errorToCloseZD0220
			#693 panFilterFailToRegen020203 <= filterFailToRegen020203
			#694 panErrorToOpenZD0215 <= errorToOpenZD0215
			#695 panErrorToCloseZD0215 <= errorToCloseZD0215
			#696 panErrorToOpenZD0221 <= errorToOpenZD0221
			#697 panErrorToCloseZD0221 <= errorToCloseZD0221
			#698 panFilterFailToRegen020204 <= filterFailToRegen020204
			#699 panErrorToOpenZD0216 <= errorToOpenZD0216
		END_MACRO
		#700 MACRO 8 bit output module 15()
			#701 panErrorToCloseZD0216 <= errorToCloseZD0216
			#702 panErrorToOpenZD0222 <= errorToOpenZD0222
			#703 panErrorToCloseZD0222 <= errorToCloseZD0222
			#704 panFilterFailToRegen020205 <= filterFailToRegen020205
			#705 panErrorToOpenZD0217 <= errorToOpenZD0217
			#706 panErrorToCloseZD0217 <= errorToCloseZD0217
			#707 panErrorToOpenZD0223 <= errorToOpenZD0223
			#708 panErrorToCloseZD0223 <= errorToCloseZD0223
		END_MACRO
		#709 MACRO 8 bit output module 16()
			#710 panFilterFailToRegen020206 <= filterFailToRegen020206
			#711 panErrorToOpenZD0218 <= errorToOpenZD0218
			#712 panErrorToCloseZD0218 <= errorToCloseZD0218
			#713 panErrorToOpenZD0224 <= errorToOpenZD0224
			#714 panErrorToCloseZD0224 <= errorToCloseZD0224
			#715 panAlarmPLKnetwork <= alarmPLKnetwork
			#716 panAlarmND050201 <= alarmND050201
			#717 panAlarmND050202 <= alarmND050202
		END_MACRO
		#718 MACRO 8 bit output module 17()
			#719 panAlarmND060201 <= alarmND060201
			#720 panAlarmND060202 <= alarmND060202
			#721 panAlarmND060301 <= alarmND060301
			#722 panAlarmND060302 <= alarmND060302
			#723 panAlarmND070301 <= alarmND070301
			#724 panAlarmND070302 <= alarmND070302
			#725 panAlarmND080301 <= alarmND080301
			#726 panAlarmND080302 <= alarmND080302
		END_MACRO
		#727 MACRO 8 bit output module 18()
			#728 panAlarmND0804 <= alarmND0804
			#729 panAlarmOGM0104overload <= alarmOGM0104overload
			#730 panAlarmRCHV0203overload <= alarmRCHV0203overload
			#731 panAlarmN040402 <= alarmN040402
			#732 panAlarmN040401 <= alarmN040401
			#733 panAlarmM0604 <= alarmM0604
			#734 panAlarmM0702 <= alarmM0702
			#735 panAlarmM0802 <= alarmM0802
		END_MACRO
		#736 MACRO 8 bit output module 19()
			#737 panAlarmN020401 <= alarmN020401
			#738 panAlarmN020402 <= alarmN020402
			#739 panAlarmFS020101 <= alarmFS020101
			#740 panAlarmFS020102 <= alarmFS020102
			#741 panAlarmFS020103 <= alarmFS020103
			#742 panAlarmFS020104 <= alarmFS020104
			#743 panAlarmFS020105 <= alarmFS020105
			#744 panAlarmFS020106 <= alarmFS020106
		END_MACRO
		#745 MACRO 8 bit output module 20()
			#746 panAlarmFS020201 <= alarmFS020201
			#747 panAlarmFS020202 <= alarmFS020202
			#748 panAlarmFS020203 <= alarmFS020203
			#749 panAlarmFS020204 <= alarmFS020204
			#750 panAlarmFS020205 <= alarmFS020205
			#751 panAlarmFS020206 <= alarmFS020206
			#752 panAlarmZDE0201power <= alarmZDE0201power
			#753 panAlarmZDE0202power <= alarmZDE0202power
		END_MACRO
		#754 MACRO 8 bit output module 21()
			#755 panAlarmZDE0203power <= alarmZDE0203power
			#756 panAlarmZDE0204power <= alarmZDE0204power
			#757 panAlarmZDE0205power <= alarmZDE0205power
			#758 panAlarmZDE0206power <= alarmZDE0206power
			#759 panAlarmZDE0207power <= alarmZDE0207power
			#760 panAlarmZDE0208power <= alarmZDE0208power
			#761 panAlarmZDE0209power <= alarmZDE0209power
			#762 panAlarmZDE0210power <= alarmZDE0210power
		END_MACRO
		#763 MACRO 8 bit output module 22()
			#764 panAlarmZDE0211power <= alarmZDE0211power
			#765 panAlarmZDE0212power <= alarmZDE0212power
			#766 panAlarmZDE0213power <= alarmZDE0213power
			#767 panAlarmZDE0214power <= alarmZDE0214power
			#768 panAlarmZDE0215power <= alarmZDE0215power
			#769 panAlarmZDE0216power <= alarmZDE0216power
			#770 panAlarmZDE0217power <= alarmZDE0217power
			#771 panAlarmZDE0218power <= alarmZDE0218power
		END_MACRO
		#772 MACRO 8 bit output module 23()
			#773 panAlarmZDE0219power <= alarmZDE0219power
			#774 panAlarmZDE0220power <= alarmZDE0220power
			#775 panAlarmZDE0221power <= alarmZDE0221power
			#776 panAlarmZDE0222power <= alarmZDE0222power
			#777 panAlarmZDE0223power <= alarmZDE0223power
			#778 panAlarmZDE0224power <= alarmZDE0224power
			#779 panAlarmZDE0225power <= alarmZDE0225power
			#780 panAlarmKSHE0401power <= alarmKSHE0401power
		END_MACRO
		#781 MACRO 8 bit output module 24()
			#782 panAlarmKNS <= alarmKNS
			#783 panAlarmPowerSocketFS <= alarmPowerSocketFS
			#784 panAlarmKEMvalvesPower <= alarmKEMvalvesPower
			#785 panAlarmEmergencyPressed <= alarmEmergencyPressed
			#786 panAlarmRKF <= alarmRKF
			#787 panUFO0301noFlowAttention <= UFO0301noFlowAttention
			#788 panM0604attention <= M0604attention
			#789 panM0702attention <= M0702attention
		END_MACRO
		#790 MACRO 8 bit output module 25()
			#791 panM0802attention <= M0802attention
			#792 panStatusKNS <= DD6_DI.8
			#793 panND0502statRegimeP1M <= ND0502statRegimeP1M
			#794 panND0502statRegimeP2M <= ND0502statRegimeP2M
			#795 panND0502statRegimeByC <= ND0502statRegimeByC
			#796 panND0502statRegimeByWT <= ND0502statRegimeByWT
			#797 panND0602statRegimeP1M <= ND0602statRegimeP1M
			#798 panND0602statRegimeP2M <= ND0602statRegimeP2M
		END_MACRO
		#799 MACRO 8 bit output module 26()
			#800 panND0602statRegimeByC <= ND0602statRegimeByC
			#801 panND0602statRegimeByWT <= ND0602statRegimeByWT
			#802 panND0603statRegimeP1M <= ND0603statRegimeP1M
			#803 panND0603statRegimeP2M <= ND0603statRegimeP2M
			#804 panND0603statRegimeByC <= ND0603statRegimeByC
			#805 panND0603statRegimeByWT <= ND0603statRegimeByWT
			#806 panND0703statRegimeP1M <= ND0703statRegimeP1M
			#807 panND0703statRegimeP2M <= ND0703statRegimeP2M
		END_MACRO
		#808 MACRO 8 bit output module 27()
			#809 panND0703statRegimeByC <= ND0703statRegimeByC
			#810 panND0703statRegimeByWT <= ND0703statRegimeByWT
			#811 panND0803statRegimeP1M <= ND0803statRegimeP1M
			#812 panND0803statRegimeP2M <= ND0803statRegimeP2M
			#813 panND0803statRegimeByC <= ND0803statRegimeByC
			#814 panND0803statRegimeByWT <= ND0803statRegimeByWT
			#815 panN0105statRegimeP1M <= N0105statRegimeP1M
			#816 panN0105statRegimeP2M <= N0105statRegimeP2M
		END_MACRO
		#817 MACRO 8 bit output module 28()
			#818 panN0105statRegimeByC <= N0105statRegimeByC
			#819 panN0105statRegimeByWT <= N0105statRegimeByWT
			#820 panN0204statRegimeP1M <= N0204statRegimeP1M
			#821 panN0204statRegimeP2M <= N0204statRegimeP2M
			#822 panN0204statRegimeByC <= N0204statRegimeByC
			#823 panN0204statRegimeWT <= N0204statRegimeWT
			#824 panN0404statRegimeP1M <= N0404statRegimeP1M
			#825 panN0404statRegimeP2M <= N0404statRegimeP2M
		END_MACRO
		#826 MACRO 8 bit output module 29()
			#827 panN0404statRegimeByC <= N0404statRegimeByC
			#828 panN0404statRegimeWT <= N0404statRegimeWT
			#829 panUFO0301statRegimeP1M <= UFO0301statRegimeP1M
			#830 panUFO0301statRegimeP2M <= UFO0301statRegimeP2M
			#831 panUFO0301statRegimeByC <= UFO0301statRegimeByC
			#832 panUFO0301statRegimeWT <= UFO0301statRegimeWT
			#833 panZDE0225open <= DD9_DI.0
			#834 panZDE0201open <= DD7_DI.16
		END_MACRO
		#835 MACRO 8 bit output module 30()
			#836 panZDE0201close <= DD7_DI.17
			#837 panZDE0202open <= DD7_DI.18
			#838 panZDE0202close <= DD7_DI.19
			#839 panZDE0203open <= DD7_DI.20
			#840 panZDE0203close <= DD7_DI.21
			#841 panZDE0204open <= DD7_DI.22
			#842 panZDE0204close <= DD7_DI.23
			#843 panZDE0205open <= DD7_DI.24
		END_MACRO
		#844 MACRO 8 bit output module 31()
			#845 panZDE0205close <= DD7_DI.25
			#846 panZDE0206open <= DD7_DI.26
			#847 panZDE0206close <= DD7_DI.27
			#848 panZDE0207open <= DD7_DI.28
			#849 panZDE0207close <= DD7_DI.29
			#850 panZDE0208open <= DD7_DI.30
			#851 panZDE0208close <= DD7_DI.31
			#852 panZDE0209open <= DD8_DI.0
		END_MACRO
		#853 MACRO 8 bit output module 32()
			#854 panZDE0209close <= DD8_DI.1
			#855 panZDE0210open <= DD8_DI.2
			#856 panZDE0210close <= DD8_DI.3
			#857 panZDE0211open <= DD8_DI.4
			#858 panZDE0211close <= DD8_DI.5
			#859 panZDE0212open <= DD8_DI.6
			#860 panZDE0212close <= DD8_DI.7
			#861 panZDE0213open <= DD8_DI.8
		END_MACRO
		#862 MACRO 8 bit output module 33()
			#863 panZDE0213close <= DD8_DI.9
			#864 panZDE0214open <= DD8_DI.10
			#865 panZDE0214close <= DD8_DI.11
			#866 panZDE0215open <= DD8_DI.12
			#867 panZDE0215close <= DD8_DI.13
			#868 panZDE0216open <= DD8_DI.14
			#869 panZDE0216close <= DD8_DI.15
			#870 panZDE0217open <= DD8_DI.16
		END_MACRO
		#871 MACRO 8 bit output module 34()
			#872 panZDE0217close <= DD8_DI.17
			#873 panZDE0218open <= DD8_DI.18
			#874 panZDE0218close <= DD8_DI.19
			#875 panZDE0219open <= DD8_DI.20
			#876 panZDE0219close <= DD8_DI.21
			#877 panZDE0220open <= DD8_DI.22
			#878 panZDE0220close <= DD8_DI.23
			#879 panZDE0221open <= DD8_DI.24
		END_MACRO
		#880 MACRO 8 bit output module 35()
			#881 panZDE0221close <= DD8_DI.25
			#882 panZDE0222open <= DD8_DI.26
			#883 panZDE0222close <= DD8_DI.27
			#884 panZDE0223open <= DD8_DI.28
			#885 panZDE0223close <= DD8_DI.29
			#886 panZDE0224open <= DD8_DI.30
			#887 panZDE0224close <= DD8_DI.31
			#888 panZDE0225close <= DD9_DI.1
		END_MACRO
		#889 MACRO 8 bit output module 36x()
			#890 panKSHE0401close <= DD9_DI.3
			#891 panZDE0301open <= DD1_DI12
			#892 panZDE0301close <= DD1_DI13
			#893 panZDE0302open <= DD1_DI14
			#894 panZDE0302close <= DD1_DI15
			#895 panErrorToOpenZDE0301 <= errorToOpenZDE0301
			#896 panErrorToCloseZDE0301 <= errorToCloseZDE0301
			#897 panErrorToOpenZDE0302 <= errorToOpenZDE0302
		END_MACRO
		#898 panErrorToCloseZDE0302 <= errorToCloseZDE0302
		#899 panAlarmZDE0301power <= alarmZDE0301power
		#900 panAlarmZDE0302power <= alarmZDE0302power
	END_MACRO
	#901 MACRO PFW регистры на чтение из панели (управление ПЛК)()
		#902 MUL(panTimeToOpenCloseValve, 1000)
		#903 REAL_TO_TIME(#902)
		#904 TimeToOpenCloseValve <= #903
		#905 maxTemperature <= panMaxTemperature
		#906 minTemperature <= panMinTemperature
		#907 ND0502setMaxDosVal <= panND0502setMaxDosVal
		#908 ND0502setKoefProp <= panND0502setKoefProp
		#909 ND0602setMaxDosVal <= panND0602setMaxDosVal
		#910 ND0602setKoefProp <= panND0602setKoefProp
		#911 ND0603setMaxDosVal <= panND0603setMaxDosVal
		#912 ND0603setKoefProp <= panND0603setKoefProp
		#913 ND0703pHsetValue <= panND0703pHsetValue
		#914 ND0703YoutManual <= panND0703YoutManual
		#915 ND0703koeffI <= panND0703koeffI
		#916 ND0703koeffD <= panND0703koeffD
		#917 ND0703koeffP <= panND0703koeffP
		#918 ND0803setMaxDosVal <= panND0803setMaxDosVal
		#919 ND0803setKoefProp <= panND0803setKoefProp
		#920 ND0804doseValue <= panND0804doseValue
		#921 N0105flowSetValue <= panN0105flowSetValue
		#922 N0105YoutManual <= panN0105YoutManual
		#923 N0105koeffI <= panN0105koeffI
		#924 N0105koeffD <= panN0105koeffD
		#925 N0105koeffP <= panN0105koeffP
		#926 FQS0301impulsValue <= panFQS0301impulsValue
		#927 FQS0301correction <= panFQS0301correction
		#928 MUL(panFPKtimeToWork, 1000)
		#929 REAL_TO_TIME(#928)
		#930 FPKtimeToWork <= #929
		#931 MUL(panFPKnotStartedTime, 1000)
		#932 REAL_TO_TIME(#931)
		#933 FPKnotStartedTime <= #932
		#934 FPKmaxPressureValue <= panFPKmaxPressureValue
		#935 filterValueToRegen <= panFilterValueToRegen
	END_MACRO
	#936 MACRO PSB регистры на чтение из панели (управление ПЛК)()
		(* PSB регистры на чтение из панели (управление ПЛК) *)
		#937 MACRO 8 bit input module 1()
			#1265 alarmReset <= panAlarmResetButton
			#1266 ND0502resetCountP1 <= panND0502resetCountP1
			#1267 ND0502resetCountP2 <= panND0502resetCountP2
			#1268 ND0502resetWorkTimeP1 <= panND0502resetWorkTimeP1
			#1269 ND0502resetWorkTimeP2 <= panND0502resetWorkTimeP2
			#1270 ND0502regimeP1M <= panND0502regimeP1M
			#1271 ND0502regimeP2M <= panND0502regimeP2M
			#1272 ND0502regimeByC <= panND0502regimeByC
		END_MACRO
		#938 MACRO 8 bit input module 2()
			#1273 ND0502regimeByWT <= panND0502regimeByWT
			#1274 ND0602resetCountP1 <= panND0602resetCountP1
			#1275 ND0602resetCountP2 <= panND0602resetCountP2
			#1276 ND0602resetWorkTimeP1 <= panND0602resetWorkTimeP1
			#1277 ND0602resetWorkTimeP2 <= panND0602resetWorkTimeP2
			#1278 ND0602regimeP1M <= panND0602regimeP1M
			#1279 ND0602regimeP2M <= panND0602regimeP2M
			#1280 ND0602regimeByC <= panND0602regimeByC
		END_MACRO
		#939 MACRO 8 bit input module 3()
			#1281 ND0602regimeByWT <= panND0602regimeByWT
			#1282 ND0603resetCountP1 <= panND0603resetCountP1
			#1283 ND0603resetCountP2 <= panND0603resetCountP2
			#1284 ND0603resetWorkTimeP1 <= panND0603resetWorkTimeP1
			#1285 ND0603resetWorkTimeP2 <= panND0603resetWorkTimeP2
			#1286 ND0603regimeP1M <= panND0603regimeP1M
			#1287 ND0603regimeP2M <= panND0603regimeP2M
			#1288 ND0603regimeByC <= panND0603regimeByC
		END_MACRO
		#940 MACRO 8 bit input module 4()
			#1289 ND0603regimeByWT <= panND0603regimeByWT
			#1290 ND0703resetCountP1 <= panND0703resetCountP1
			#1291 ND0703resetCountP2 <= panND0703resetCountP2
			#1292 ND0703resetWorkTimeP1 <= panND0703resetWorkTimeP1
			#1293 ND0703resetWorkTimeP2 <= panND0703resetWorkTimeP2
			#1294 ND0703regimeP1M <= panND0703regimeP1M
			#1295 ND0703regimeP2M <= panND0703regimeP2M
			#1296 ND0703regimeByC <= panND0703regimeByC
		END_MACRO
		#941 MACRO 8 bit input module 5()
			#1297 ND0703regimeByWT <= panND0703regimeByWT
			#1298 ND0703YmanAuto <= panND0703YmanAuto
			#1299 ND0803resetCountP1 <= panND0803resetCountP1
			#1300 ND0803resetCountP2 <= panND0803resetCountP2
			#1301 ND0803resetWorkTimeP1 <= panND0803resetWorkTimeP1
			#1302 ND0803resetWorkTimeP2 <= panND0803resetWorkTimeP2
			#1303 ND0803regimeP1M <= panND0803regimeP1M
			#1304 ND0803regimeP2M <= panND0803regimeP2M
		END_MACRO
		#942 MACRO 8 bit input module 6()
			#1305 ND0803regimeByC <= panND0803regimeByC
			#1306 ND0803regimeByWT <= panND0803regimeByWT
			#1307 N0105resetCountP1 <= panN0105resetCountP1
			#1308 N0105resetCountP2 <= panN0105resetCountP2
			#1309 N0105resetWorkTimeP1 <= panN0105resetWorkTimeP1
			#1310 N0105resetWorkTimeP2 <= panN0105resetWorkTimeP2
			#1311 N0105regimeByC <= panN0105regimeByC
			#1312 N0105regimeByWT <= panN0105regimeByWT
		END_MACRO
		#943 MACRO 8 bit input module 7()
			#1313 N0105YmanAuto <= panN0105YmanAuto
			#1314 N0204resetCountP1 <= panN0204resetCountP1
			#1315 N0204resetCountP2 <= panN0204resetCountP2
			#1316 N0204resetWorkTimeP1 <= panN0204resetWorkTimeP1
			#1317 N0204resetWorkTimeP2 <= panN0204resetWorkTimeP2
			#1318 N0204regimeP1M <= panN0204regimeP1M
			#1319 N0204regimeP2M <= panN0204regimeP2M
			#1320 N0204regimeByC <= panN0204regimeByC
		END_MACRO
		#944 MACRO 8 bit input module 8()
			#1321 N0204regimeWT <= panN0204regimeWT
			#1322 UFO0301resetCountP1 <= panUFO0301resetCountP1
			#1323 UFO0301resetCountP2 <= panUFO0301resetCountP2
			#1324 UFO0301resetWorkTimeP1 <= panUFO0301resetWorkTimeP1
			#1325 UFO0301resetWorkTimeP2 <= panUFO0301resetWorkTimeP2
			#1326 UFO0301regimeP1M <= panUFO0301regimeP1M
			#1327 UFO0301regimeP2M <= panUFO0301regimeP2M
			#1328 UFO0301regimeByC <= panUFO0301regimeByC
		END_MACRO
		#945 MACRO 8 bit input module 9()
			#1329 UFO0301regimeWT <= panUFO0301regimeWT
			#1330 N0404resetCountP1 <= panN0404resetCountP1
			#1331 N0404resetCountP2 <= panN0404resetCountP2
			#1332 N0404resetWorkTimeP1 <= panN0404resetWorkTimeP1
			#1333 N0404resetWorkTimeP2 <= panN0404resetWorkTimeP2
			#1334 N0404regimeP1M <= panN0404regimeP1M
			#1335 N0404regimeP2M <= panN0404regimeP2M
			#1336 N0404regimeByC <= panN0404regimeByC
		END_MACRO
		#946 MACRO 8 bit input module 10-11()
			(* одули 10 и 11 заполнены переменными для тестирования задвижек. / Здесь они не показаны, т.к. спешка. / Они вставлены напрямую в макросы управления промывкой фильтров. / testValvesFS020101 - testValvesFS020206 (PSB612-623) *)
			#1337 N0404regimeWT <= panN0404regimeWT
			#1338 FQS0301reset <= panFQS0301reset
			#1339 FQS0301addCorrection <= panFQS0301addCorrection
			#1340 FQS0301deleteCorrection <= panFQS0301deleteCorrection
		END_MACRO
		#947 testKSHE0401 <= panTestKSHE0401
		#948 testZDE0225 <= panTestZDE0225
		#949 testZDE03 <= panTestZDE03
		#950 manualZDE0301 <= panManualZDE0301
		#951 manualZDE0302 <= panManualZDE0302
	END_MACRO
END_MACRO
#952 NOT(DD6_DI.13)
#953 alarmRCHV0203overload <= #952
#954 NOT(DD9_DI.5)
#955 alarmZDE0202power <= #954
#956 NOT(DD9_DI.26)
#957 alarmZDE0223power <= #956
#958 MACRO переменные на диспетчеризацию()
	#959 remFT0101value <= DD1_AI1_FT0101value
	#960 remFQS0301totalAmount <= FQS0301totalAmount
	#961 remTemperatureValue <= temperatureValue
	#962 remStatusN010501started <= N0105statStartedP1
	#963 remStatusN010502started <= N0105statStartedP2
	#964 remStatusUFO030101started <= DD5_DI.26
	#965 remStatusUFO030102started <= DD5_DI.28
	#966 remAlarm <= Alarm
	#967 remN010501alarm <= N010501alarm
	#968 remN010502alarm <= N010502alarm
	#969 remFPKalarm <= DD7_DI.14
	#970 remUFO030101alarm <= DD5_DI.27
	#971 remUFO030102alarm <= DD5_DI.29
	#972 remAlarmEmergencyPressed <= alarmEmergencyPressed
	#973 remAlarmOOGM0104overload <= DD6_DI.11
	#974 remAlarmRCHV0203overload <= DD6_DI.13
END_MACRO
#975 NOT(DD5_DI.14)
#976 alarmN040402 <= #975
#977 NOT(DD9_DI.6)
#978 alarmZDE0203power <= #977
#979 NOT(DD9_DI.27)
#980 alarmZDE0224power <= #979
#981 NOT(DD5_DI.15)
#982 alarmN040401 <= #981
#983 NOT(DD9_DI.7)
#984 alarmZDE0204power <= #983
#985 NOT(DD9_DI.28)
#986 alarmZDE0225power <= #985
#987 NOT(DD5_DI.20)
#988 alarmM0604 <= #987
#989 NOT(DD9_DI.8)
#990 alarmZDE0205power <= #989
#991 NOT(DD9_DI.29)
#992 alarmKSHE0401power <= #991
#993 NOT(DD5_DI.22)
#994 alarmM0702 <= #993
#995 NOT(DD9_DI.9)
#996 alarmZDE0206power <= #995
#997 NOT(DD6_DI.9)
#998 alarmKNS <= #997
#999 NOT(DD5_DI.24)
#1000 alarmM0802 <= #999
#1001 NOT(DD9_DI.10)
#1002 alarmZDE0207power <= #1001
#1003 NOT(DD6_DI.17)
#1004 alarmPowerSocketFS <= #1003
#1005 NOT(DD5_DI.7)
#1006 alarmN020401 <= #1005
#1007 NOT(DD9_DI.11)
#1008 alarmZDE0208power <= #1007
#1009 NOT(DD6_DI.18)
#1010 alarmKEMvalvesPower <= #1009
#1011 NOT(DD5_DI.8)
#1012 alarmN020402 <= #1011
#1013 NOT(DD9_DI.12)
#1014 alarmZDE0209power <= #1013
#1015 NOT(DD1_DI4)
#1016 alarmEmergencyPressed <= #1015
#1017 GT(DD1_AI2_FT0102value, 0)
#1018 filterPulserGen:PulsePerSec(start: #1017)
#1019 DIV(DD1_AI2_FT0102value, 3600)
#1020 ADD(EN: #1018.out, #1019, filterTotalAmountFT0102)
#1021 filterTotalAmountFT0102 <= #1020
#1022 NOT(DD6_DI.21)
#1023 alarmFS020101 <= #1022
#1024 NOT(DD9_DI.13)
#1025 alarmZDE0210power <= #1024
#1026 NOT(DD1_DI5)
#1027 alarmRKF <= #1026
#1028 NOT(DD9_DI.30)
#1029 alarmZDE0301power <= #1028
#1030 NOT(DD9_DI.31)
#1031 alarmZDE0302power <= #1030
#1032 MOVE(EN: filterTotalAmountReset, 0)
#1033 filterTotalAmountFT0102 <= #1032
#1034 GE(filterTotalAmountFT0102, filterValueToRegen)
#1035 MACRO управление промывкой фильтра ФС02.01.01(pin 1 "сигнал на промывку": #1034, pin 2 "авария фильтра": DD6_DI.21, pin 3 "подтверждение промывки": DD6_DI.20, pin 4 "сброс аварий": alarmReset, pin 5 "начать очередь снова": filterStartNewQueue, pin 6 "ЗДЭ02.01 открыта": DD7_DI.16, pin 7 "ЗДЭ02.01 закрыта": DD7_DI.17, pin 8 "ЗДЭ02.07 открыта": DD7_DI.28, pin 9 "ЗДЭ02.07 закрыта": DD7_DI.29, pin 10 "время движения ЗДЭ": timeToOpenCloseValve, pin 11 "авария питания ЗДЭ02.01": DD9_DI.4, pin 12 "авария питания ЗДЭ02.07": DD9_DI.10)
	(* если открыт = фильтрация *)
	(* если открыт = промывка *)
	(* <- выход использовать в / последнем фильтре для / начала очереди заново *)
	out 1 "следующий в очереди" <= #1038.output
	out 2 "промыть ФС02.01.01" <= #1037
	#1036 ZD0201:SimpleValve(inputOpen: NOT #1037, inputClose: #1037, statusOpen: pin 6, statusClose: pin 7, reset: pin 4, timeToOpenClose: pin 10)
	out 6 "открыть ЗДЭ02.01" <= #1036.outputOpen
	out 7 "закрыть ЗДЭ02.01" <= #1036.outputClose
	out 8 "авария открытия ЗДЭ02.01" <= #1036.errorToOpen
	#1037 OR(panTestValvesFS020101, #1038.regenFilterOUT)
	out 9 "авария закрытия ЗДЭ02.01" <= #1036.errorToClose
	#1038 FS020101manager:FilterQueueManager(input: pin 1, filterAlarm: #1039, regenFilterStatus: pin 3, alarmReset: pin 4, startNextLoop: pin 5)
	#1039 OR(alarmZD020107, pin 2, pin 11, pin 12)
	out 3 "ФС02.01.01 промыт" <= #1038.regenerated
	out 4 "не удалось промыть" <= #1038.failToRegen
	#1040 OR(#1036.errorToOpen, #1036.errorToClose, #1042.errorToOpen, #1042.errorToClose)
	#1041 alarmZD020107 <= #1040
	out 5 "сброс счетчика" <= #1038.counterReset
	#1042 ZD0207:SimpleValve(inputOpen: #1037, inputClose: NOT #1037, statusOpen: pin 8, statusClose: pin 9, reset: pin 4, timeToOpenClose: pin 10)
	out 10 "открыть ЗДЭ02.07" <= #1042.outputOpen
	out 11 "закрыть ЗДЭ02.07" <= #1042.outputClose
	out 12 "авария открытия ЗДЭ02.07" <= #1042.errorToOpen
	out 13 "авария закрытия ЗДЭ02.07" <= #1042.errorToClose
END_MACRO
#1043 DD2_DO.4 <= #1035.out 2
#1044 regeneratedFS020101 <= #1035.out 3
#1045 filterFailToRegen020101 <= #1035.out 4
#1046 filterTotalAmountReset <= #1035.out 5
#1047 DD2_DO.16 <= #1035.out 6
#1048 DD2_DO.17 <= #1035.out 7
#1049 errorToOpenZD0201 <= #1035.out 8
#1050 errorToCloseZD0201 <= #1035.out 9
#1051 DD2_DO.28 <= #1035.out 10
#1052 DD2_DO.29 <= #1035.out 11
#1053 errorToOpenZD0207 <= #1035.out 12
#1054 errorToCloseZD0207 <= #1035.out 13
#1055 MACRO управление промывкой фильтра ФС02.01.02(pin 1 "сигнал на промывку": #1035.out 1, pin 2 "авария фильтра": DD6_DI.23, pin 3 "подтверждение промывки": DD6_DI.22, pin 4 "сброс аварий": alarmReset, pin 5 "начать очередь снова": filterStartNewQueue, pin 6 "ЗДЭ02.02 открыта": DD7_DI.18, pin 7 "ЗДЭ02.02 закрыта": DD7_DI.19, pin 8 "ЗДЭ02.08 открыта": DD7_DI.30, pin 9 "ЗДЭ02.08 закрыта": DD7_DI.31, pin 10 "время движения ЗДЭ": timeToOpenCloseValve, pin 11 "авария питания ЗДЭ02.02": DD9_DI.5, pin 12 "авария питания ЗДЭ02.08": DD9_DI.11)
	(* если открыт = фильтрация *)
	(* если открыт = промывка *)
	(* <- выход использовать в / последнем фильтре для / начала очереди заново *)
	out 1 "следующий в очереди" <= #1058.output
	out 2 "промыть ФС02.01.02" <= #1057
	#1056 ZD0202:SimpleValve(inputOpen: NOT #1057, inputClose: #1057, statusOpen: pin 6, statusClose: pin 7, reset: pin 4, timeToOpenClose: pin 10)
	out 5 "открыть ЗДЭ02.02" <= #1056.outputOpen
	out 6 "закрыть ЗДЭ02.02" <= #1056.outputClose
	out 7 "авария открытия ЗДЭ02.02" <= #1056.errorToOpen
	#1057 OR(panTestValvesFS020102, #1058.regenFilterOUT)
	out 8 "авария закрытия ЗДЭ02.02" <= #1056.errorToClose
	#1058 FS020102manager:FilterQueueManager(input: pin 1, filterAlarm: #1059, regenFilterStatus: pin 3, alarmReset: pin 4, startNextLoop: pin 5)
	#1059 OR(alarmZD020208, pin 2, pin 11, pin 12)
	#1060 OR(#1056.errorToOpen, #1056.errorToClose, #1062.errorToOpen, #1062.errorToClose)
	#1061 alarmZD020208 <= #1060
	out 3 "ФС02.01.02 промыт" <= #1058.regenerated
	out 4 "не удалось промыть" <= #1058.failToRegen
	#1062 ZD0208:SimpleValve(inputOpen: #1057, inputClose: NOT #1057, statusOpen: pin 8, statusClose: pin 9, reset: pin 4, timeToOpenClose: pin 10)
	out 9 "открыть ЗДЭ02.08" <= #1062.outputOpen
	out 10 "закрыть ЗДЭ02.08" <= #1062.outputClose
	out 11 "авария открытия ЗДЭ02.08" <= #1062.errorToOpen
	out 12 "авария закрытия ЗДЭ02.08" <= #1062.errorToClose
END_MACRO
#1063 DD2_DO.5 <= #1055.out 2
#1064 regeneratedFS020102 <= #1055.out 3
#1065 filterFailToRegen020102 <= #1055.out 4
#1066 DD2_DO.18 <= #1055.out 5
#1067 DD2_DO.19 <= #1055.out 6
#1068 errorToOpenZD0202 <= #1055.out 7
#1069 errorToCloseZD0202 <= #1055.out 8
#1070 DD2_DO.30 <= #1055.out 9
#1071 DD2_DO.31 <= #1055.out 10
#1072 errorToOpenZD0208 <= #1055.out 11
#1073 errorToCloseZD0208 <= #1055.out 12
#1074 MACRO управление промывкой фильтра ФС02.01.03(pin 1 "сигнал на промывку": #1055.out 1, pin 2 "авария фильтра": DD6_DI.25, pin 3 "подтверждение промывки": DD6_DI.24, pin 4 "сброс аварий": alarmReset, pin 5 "начать очередь снова": filterStartNewQueue, pin 6 "ЗДЭ02.03 открыта": DD7_DI.20, pin 7 "ЗДЭ02.03 закрыта": DD7_DI.21, pin 8 "ЗДЭ02.09 открыта": DD8_DI.0, pin 9 "ЗДЭ02.09 закрыта": DD8_DI.1, pin 10 "время движения ЗДЭ": timeToOpenCloseValve, pin 11 "авария питания ЗДЭ02.03": DD9_DI.6, pin 12 "авария питания ЗДЭ02.09": DD9_DI.12)
	(* если открыт = фильтрация *)
	(* если открыт = промывка *)
	(* <- выход использовать в / последнем фильтре для / начала очереди заново *)
	out 1 "следующий в очереди" <= #1077.output
	out 2 "промыть ФС02.01.03" <= #1076
	#1075 ZD0203:SimpleValve(inputOpen: NOT #1076, inputClose: #1076, statusOpen: pin 6, statusClose: pin 7, reset: pin 4, timeToOpenClose: pin 10)
	out 5 "открыть ЗДЭ02.03" <= #1075.outputOpen
	out 6 "закрыть ЗДЭ02.03" <= #1075.outputClose
	out 7 "авария открытия ЗДЭ02.03" <= #1075.errorToOpen
	#1076 OR(panTestValvesFS020103, #1077.regenFilterOUT)
	out 8 "авария закрытия ЗДЭ02.03" <= #1075.errorToClose
	#1077 FS020103manager:FilterQueueManager(input: pin 1, filterAlarm: #1078, regenFilterStatus: pin 3, alarmReset: pin 4, startNextLoop: pin 5)
	#1078 OR(alarmZD020309, pin 2, pin 11, pin 12)
	#1079 OR(#1075.errorToOpen, #1075.errorToClose, #1081.errorToOpen, #1081.errorToClose)
	#1080 alarmZD020309 <= #1079
	out 3 "ФС02.01.03 промыт" <= #1077.regenerated
	out 4 "не удалось промыть" <= #1077.failToRegen
	#1081 ZD0209:SimpleValve(inputOpen: #1076, inputClose: NOT #1076, statusOpen: pin 8, statusClose: pin 9, reset: pin 4, timeToOpenClose: pin 10)
	out 9 "открыть ЗДЭ02.09" <= #1081.outputOpen
	out 10 "закрыть ЗДЭ02.09" <= #1081.outputClose
	out 11 "авария открытия ЗДЭ02.09" <= #1081.errorToOpen
	out 12 "авария закрытия ЗДЭ02.09" <= #1081.errorToClose
END_MACRO
#1082 DD2_DO.6 <= #1074.out 2
#1083 regeneratedFS020103 <= #1074.out 3
#1084 filterFailToRegen020103 <= #1074.out 4
#1085 DD2_DO.20 <= #1074.out 5
#1086 DD2_DO.21 <= #1074.out 6
#1087 errorToOpenZD0203 <= #1074.out 7
#1088 errorToCloseZD0203 <= #1074.out 8
#1089 DD3_DO.0 <= #1074.out 9
#1090 DD3_DO.1 <= #1074.out 10
#1091 errorToOpenZD0209 <= #1074.out 11
#1092 errorToCloseZD0209 <= #1074.out 12
#1093 MACRO управление промывкой фильтра ФС02.01.04(pin 1 "сигнал на промывку": #1074.out 1, pin 2 "авария фильтра": DD6_DI.27, pin 3 "подтверждение промывки": DD6_DI.26, pin 4 "сброс аварий": alarmReset, pin 5 "начать очередь снова": filterStartNewQueue, pin 6 "ЗДЭ02.04 открыта": DD7_DI.22, pin 7 "ЗДЭ02.04 закрыта": DD7_DI.23, pin 8 "ЗДЭ02.10 открыта": DD8_DI.2, pin 9 "ЗДЭ02.10 закрыта": DD8_DI.3, pin 10 "время движения ЗДЭ": timeToOpenCloseValve, pin 11 "авария питания ЗДЭ02.04": DD9_DI.7, pin 12 "авария питания ЗДЭ02.10": DD9_DI.13)
	(* если открыт = фильтрация *)
	(* если открыт = промывка *)
	(* <- выход использовать в / последнем фильтре для / начала очереди заново *)
	out 1 "следующий в очереди" <= #1096.output
	out 2 "промыть ФС02.01.04" <= #1095
	#1094 ZD0204:SimpleValve(inputOpen: NOT #1095, inputClose: #1095, statusOpen: pin 6, statusClose: pin 7, reset: pin 4, timeToOpenClose: pin 10)
	out 5 "открыть ЗДЭ02.04" <= #1094.outputOpen
	out 6 "закрыть ЗДЭ02.04" <= #1094.outputClose
	out 7 "авария открытия ЗДЭ02.04" <= #1094.errorToOpen
	#1095 OR(panTestValvesFS020104, #1096.regenFilterOUT)
	out 8 "авария закрытия ЗДЭ02.04" <= #1094.errorToClose
	#1096 FS020104manager:FilterQueueManager(input: pin 1, filterAlarm: #1097, regenFilterStatus: pin 3, alarmReset: pin 4, startNextLoop: pin 5)
	#1097 OR(alarmZD020410, pin 2, pin 11, pin 12)
	#1098 OR(#1094.errorToOpen, #1094.errorToClose, #1100.errorToOpen, #1100.errorToClose)
	#1099 alarmZD020410 <= #1098
	out 3 "ФС02.01.04 промыт" <= #1096.regenerated
	out 4 "не удалось промыть" <= #1096.failToRegen
	#1100 ZD0210:SimpleValve(inputOpen: #1095, inputClose: NOT #1095, statusOpen: pin 8, statusClose: pin 9, reset: pin 4, timeToOpenClose: pin 10)
	out 9 "открыть ЗДЭ02.10" <= #1100.outputOpen
	out 10 "закрыть ЗДЭ02.10" <= #1100.outputClose
	out 11 "авария открытия ЗДЭ02.10" <= #1100.errorToOpen
	out 12 "авария закрытия ЗДЭ02.10" <= #1100.errorToClose
END_MACRO
#1101 DD2_DO.7 <= #1093.out 2
#1102 regeneratedFS020104 <= #1093.out 3
#1103 filterFailToRegen020104 <= #1093.out 4
#1104 DD2_DO.22 <= #1093.out 5
#1105 DD2_DO.23 <= #1093.out 6
#1106 errorToOpenZD0204 <= #1093.out 7
#1107 errorToCloseZD0204 <= #1093.out 8
#1108 DD3_DO.2 <= #1093.out 9
#1109 DD3_DO.3 <= #1093.out 10
#1110 errorToOpenZD0210 <= #1093.out 11
#1111 errorToCloseZD0210 <= #1093.out 12
#1112 MACRO управление промывкой фильтра ФС02.01.05(pin 1 "сигнал на промывку": #1093.out 1, pin 2 "авария фильтра": DD6_DI.29, pin 3 "подтверждение промывки": DD6_DI.28, pin 4 "сброс аварий": alarmReset, pin 5 "начать очередь снова": filterStartNewQueue, pin 6 "ЗДЭ02.05 открыта": DD7_DI.24, pin 7 "ЗДЭ02.05 закрыта": DD7_DI.25, pin 8 "ЗДЭ02.11 открыта": DD8_DI.4, pin 9 "ЗДЭ02.11 закрыта": DD8_DI.5, pin 10 "время движения ЗДЭ": timeToOpenCloseValve, pin 11 "авария питания ЗДЭ02.05": DD9_DI.8, pin 12 "авария питания ЗДЭ02.11": DD9_DI.14)
	(* если открыт = фильтрация *)
	(* если открыт = промывка *)
	(* <- выход использовать в / последнем фильтре для / начала очереди заново *)
	out 1 "следующий в очереди" <= #1115.output
	out 2 "промыть ФС02.01.05" <= #1114
	#1113 ZD0205:SimpleValve(inputOpen: NOT #1114, inputClose: #1114, statusOpen: pin 6, statusClose: pin 7, reset: pin 4, timeToOpenClose: pin 10)
	out 5 "открыть ЗДЭ02.05" <= #1113.outputOpen
	out 6 "закрыть ЗДЭ02.05" <= #1113.outputClose
	out 7 "авария открытия ЗДЭ02.05" <= #1113.errorToOpen
	#1114 OR(panTestValvesFS020105, #1115.regenFilterOUT)
	out 8 "авария закрытия ЗДЭ02.05" <= #1113.errorToClose
	#1115 FS020105manager:FilterQueueManager(input: pin 1, filterAlarm: #1116, regenFilterStatus: pin 3, alarmReset: pin 4, startNextLoop: pin 5)
	#1116 OR(alarmZD020511, pin 2, pin 11, pin 12)
	#1117 OR(#1113.errorToOpen, #1113.errorToClose, #1119.errorToOpen, #1119.errorToClose)
	#1118 alarmZD020511 <= #1117
	out 3 "ФС02.01.05 промыт" <= #1115.regenerated
	out 4 "не удалось промыть" <= #1115.failToRegen
	#1119 ZD0211:SimpleValve(inputOpen: #1114, inputClose: NOT #1114, statusOpen: pin 8, statusClose: pin 9, reset: pin 4, timeToOpenClose: pin 10)
	out 9 "открыть ЗДЭ02.11" <= #1119.outputOpen
	out 10 "закрыть ЗДЭ02.11" <= #1119.outputClose
	out 11 "авария открытия ЗДЭ02.11" <= #1119.errorToOpen
	out 12 "авария закрытия ЗДЭ02.11" <= #1119.errorToClose
END_MACRO
#1120 DD2_DO.8 <= #1112.out 2
#1121 regeneratedFS020105 <= #1112.out 3
#1122 filterFailToRegen020105 <= #1112.out 4
#1123 DD2_DO.24 <= #1112.out 5
#1124 DD2_DO.25 <= #1112.out 6
#1125 errorToOpenZD0205 <= #1112.out 7
#1126 errorToCloseZD0205 <= #1112.out 8
#1127 DD3_DO.4 <= #1112.out 9
#1128 DD3_DO.5 <= #1112.out 10
#1129 errorToOpenZD0211 <= #1112.out 11
#1130 errorToCloseZD0211 <= #1112.out 12
#1131 MACRO управление промывкой фильтра ФС02.01.06(pin 1 "сигнал на промывку": #1112.out 1, pin 2 "авария фильтра": DD6_DI.31, pin 3 "подтверждение промывки": DD6_DI.30, pin 4 "сброс аварий": alarmReset, pin 5 "начать очередь снова": filterStartNewQueue, pin 6 "ЗДЭ02.06 открыта": DD7_DI.26, pin 7 "ЗДЭ02.06 закрыта": DD7_DI.27, pin 8 "ЗДЭ02.12 открыта": DD8_DI.6, pin 9 "ЗДЭ02.12 закрыта": DD8_DI.7, pin 10 "время движения ЗДЭ": timeToOpenCloseValve, pin 11 "авария питания ЗДЭ02.06": DD9_DI.9, pin 12 "авария питания ЗДЭ02.12": DD9_DI.15)
	(* если открыт = фильтрация *)
	(* если открыт = промывка *)
	(* <- выход использовать в / последнем фильтре для / начала очереди заново *)
	out 1 "следующий в очереди" <= #1134.output
	out 2 "промыть ФС02.01.06" <= #1133
	#1132 ZD0206:SimpleValve(inputOpen: NOT #1133, inputClose: #1133, statusOpen: pin 6, statusClose: pin 7, reset: pin 4, timeToOpenClose: pin 10)
	out 5 "открыть ЗДЭ02.06" <= #1132.outputOpen
	out 6 "закрыть ЗДЭ02.06" <= #1132.outputClose
	out 7 "авария открытия ЗДЭ02.06" <= #1132.errorToOpen
	#1133 OR(panTestValvesFS020106, #1134.regenFilterOUT)
	out 8 "авария закрытия ЗДЭ02.06" <= #1132.errorToClose
	#1134 FS020106manager:FilterQueueManager(input: pin 1, filterAlarm: #1135, regenFilterStatus: pin 3, alarmReset: pin 4, startNextLoop: pin 5)
	#1135 OR(alarmZD020612, pin 2, pin 11, pin 12)
	#1136 OR(#1132.errorToOpen, #1132.errorToClose, #1138.errorToOpen, #1138.errorToClose)
	#1137 alarmZD020612 <= #1136
	out 3 "ФС02.01.06 промыт" <= #1134.regenerated
	out 4 "не удалось промыть" <= #1134.failToRegen
	#1138 ZD0212:SimpleValve(inputOpen: #1133, inputClose: NOT #1133, statusOpen: pin 8, statusClose: pin 9, reset: pin 4, timeToOpenClose: pin 10)
	out 9 "открыть ЗДЭ02.12" <= #1138.outputOpen
	out 10 "закрыть ЗДЭ02.12" <= #1138.outputClose
	out 11 "авария открытия ЗДЭ02.12" <= #1138.errorToOpen
	out 12 "авария закрытия ЗДЭ02.12" <= #1138.errorToClose
END_MACRO
#1139 DD2_DO.9 <= #1131.out 2
#1140 regeneratedFS020106 <= #1131.out 3
#1141 filterFailToRegen020106 <= #1131.out 4
#1142 DD2_DO.26 <= #1131.out 5
#1143 DD2_DO.27 <= #1131.out 6
#1144 errorToOpenZD0206 <= #1131.out 7
#1145 errorToCloseZD0206 <= #1131.out 8
#1146 DD3_DO.6 <= #1131.out 9
#1147 DD3_DO.7 <= #1131.out 10
#1148 errorToOpenZD0212 <= #1131.out 11
#1149 errorToCloseZD0212 <= #1131.out 12
#1150 MACRO управление промывкой фильтра ФС02.02.01(pin 1 "сигнал на промывку": #1131.out 1, pin 2 "авария фильтра": DD7_DI.1, pin 3 "подтверждение промывки": DD7_DI.0, pin 4 "сброс аварий": alarmReset, pin 5 "начать очередь снова": filterStartNewQueue, pin 6 "ЗДЭ02.13 открыта": DD8_DI.8, pin 7 "ЗДЭ02.13 закрыта": DD8_DI.9, pin 8 "ЗДЭ02.19 открыта": DD8_DI.20, pin 9 "ЗДЭ02.19 закрыта": DD8_DI.21, pin 10 "время движения ЗДЭ": timeToOpenCloseValve, pin 11 "авария питания ЗДЭ02.13": DD9_DI.16, pin 12 "авария питания ЗДЭ02.19": DD9_DI.22)
	(* если открыт = фильтрация *)
	(* если открыт = промывка *)
	(* <- выход использовать в / последнем фильтре для / начала очереди заново *)
	out 1 "следующий в очереди" <= #1153.output
	out 2 "промыть ФС02.02.01" <= #1152
	#1151 ZD0213:SimpleValve(inputOpen: NOT #1152, inputClose: #1152, statusOpen: pin 6, statusClose: pin 7, reset: pin 4, timeToOpenClose: pin 10)
	out 5 "открыть ЗДЭ02.13" <= #1151.outputOpen
	out 6 "закрыть ЗДЭ02.13" <= #1151.outputClose
	out 7 "авария открытия ЗДЭ02.13" <= #1151.errorToOpen
